LIN {X 0,Y 323.543,Z 923.96,A -85,B 0,C 180,E1 -15317.195,E2 -15317.195} C_VEL
LIN {X 0,Y 320.195,Z 901.46,A -85,B 0,C 180,E1 -15318.02,E2 -15318.02} C_VEL
LIN {X 0,Y 319.838,Z 896.268,A -85,B 0,C 180,E1 -15319.913,E2 -15319.913} C_VEL
LIN {X 0,Y 319.734,Z 895.469,A -85,B 0,C 180,E1 -15320.255,E2 -15320.255} C_VEL
LIN {X 0,Y 319.527,Z 895.494,A -85,B 0,C 180,E1 -15324.703,E2 -15324.703} C_VEL
LIN {X 0,Y 319.569,Z 895.487,A -85,B 0,C 180,E1 -15328.396,E2 -15328.396} C_VEL
LIN {X 0,Y 319.525,Z 895.494,A -85,B 0,C 180,E1 -15331.863,E2 -15331.863} C_VEL
LIN {X 0,Y 319.58,Z 895.491,A -85,B 0,C 180,E1 -15335.543,E2 -15335.543} C_VEL
LIN {X 0,Y 319.53,Z 895.497,A -85,B 0,C 180,E1 -15339.663,E2 -15339.663} C_VEL
LIN {X 0,Y 319.52,Z 895.495,A -85,B 0,C 180,E1 -15343.46,E2 -15343.46} C_VEL
LIN {X 0,Y 319.552,Z 895.489,A -85,B 0,C 180,E1 -15347.016,E2 -15347.016} C_VEL
LIN {X 0,Y 319.517,Z 895.498,A -85,B 0,C 180,E1 -15350.367,E2 -15350.367} C_VEL
LIN {X 0,Y 319.581,Z 895.491,A -85,B 0,C 180,E1 -15354.458,E2 -15354.458} C_VEL
LIN {X 0,Y 319.527,Z 895.494,A -85,B 0,C 180,E1 -15358.138,E2 -15358.138} C_VEL
LIN {X 0,Y 319.572,Z 895.486,A -85,B 0,C 180,E1 -15361.605,E2 -15361.605} C_VEL
LIN {X 0,Y 319.574,Z 895.488,A -85,B 0,C 180,E1 -15365.302,E2 -15365.302} C_VEL
LIN {X 0,Y 319.566,Z 895.487,A -85,B 0,C 180,E1 -15368.046,E2 -15368.046} C_VEL
LIN {X 0,Y 319.596,Z 895.483,A -85,B 0,C 180,E1 -15372.07,E2 -15372.07} C_VEL
LIN {X 0,Y 319.734,Z 895.467,A -85,B 0,C 180,E1 -15376.008,E2 -15376.008} C_VEL
LIN {X 0,Y 319.737,Z 895.469,A -85,B 0,C 180,E1 -15379.872,E2 -15379.872} C_VEL
LIN {X 0,Y 319.901,Z 895.452,A -85,B 0,C 180,E1 -15383.694,E2 -15383.694} C_VEL
LIN {X 0,Y 319.999,Z 895.433,A -85,B 0,C 180,E1 -15388.742,E2 -15388.742} C_VEL
LIN {X 0,Y 319.934,Z 895.444,A -85,B 0,C 180,E1 -15392.518,E2 -15392.518} C_VEL
LIN {X 0,Y 319.901,Z 895.452,A -85,B 0,C 180,E1 -15396.307,E2 -15396.307} C_VEL
LIN {X 0,Y 319.738,Z 895.469,A -85,B 0,C 180,E1 -15400.128,E2 -15400.128} C_VEL
LIN {X 0,Y 319.705,Z 895.471,A -85,B 0,C 180,E1 -15403.994,E2 -15403.994} C_VEL
LIN {X 0,Y 319.589,Z 895.484,A -85,B 0,C 180,E1 -15407.931,E2 -15407.931} C_VEL
LIN {X 0,Y 319.567,Z 895.487,A -85,B 0,C 180,E1 -15411.955,E2 -15411.955} C_VEL
LIN {X 0,Y 319.553,Z 895.489,A -85,B 0,C 180,E1 -15416.096,E2 -15416.096} C_VEL
LIN {X 0,Y 319.544,Z 895.493,A -85,B 0,C 180,E1 -15418.938,E2 -15418.938} C_VEL
LIN {X 0,Y 319.528,Z 895.494,A -85,B 0,C 180,E1 -15421.863,E2 -15421.863} C_VEL
LIN {X 0,Y 319.583,Z 895.491,A -85,B 0,C 180,E1 -15425.542,E2 -15425.542} C_VEL
LIN {X 0,Y 319.532,Z 895.497,A -85,B 0,C 180,E1 -15429.662,E2 -15429.662} C_VEL
LIN {X 0,Y 319.522,Z 895.494,A -85,B 0,C 180,E1 -15433.46,E2 -15433.46} C_VEL
LIN {X 0,Y 319.554,Z 895.489,A -85,B 0,C 180,E1 -15437.015,E2 -15437.015} C_VEL
LIN {X 0,Y 319.518,Z 895.498,A -85,B 0,C 180,E1 -15440.366,E2 -15440.366} C_VEL
LIN {X 0,Y 319.582,Z 895.491,A -85,B 0,C 180,E1 -15444.457,E2 -15444.457} C_VEL
LIN {X 0,Y 319.528,Z 895.494,A -85,B 0,C 180,E1 -15448.137,E2 -15448.137} C_VEL
LIN {X 0,Y 319.572,Z 895.486,A -85,B 0,C 180,E1 -15451.604,E2 -15451.604} C_VEL
LIN {X 0,Y 319.529,Z 895.494,A -85,B 0,C 180,E1 -15455.297,E2 -15455.297} C_VEL
LIN {X 0,Y 319.565,Z 895.487,A -85,B 0,C 180,E1 -15458.045,E2 -15458.045} C_VEL
LIN {X 0,Y 319.552,Z 895.489,A -85,B 0,C 180,E1 -15460.098,E2 -15460.098} C_VEL
LIN {X 0,Y 318.924,Z 895.573,A -85,B 0,C 180,E1 -15461.149,E2 -15461.149} C_VEL
LIN {X 0,Y 316.172,Z 895.918,A -85,B 0,C 180,E1 -15462.862,E2 -15462.862} C_VEL
LIN {X 0,Y 313.804,Z 896.215,A -85,B 0,C 180,E1 -15464.25,E2 -15464.25} C_VEL
LIN {X 0,Y 312.75,Z 896.342,A -85,B 0,C 180,E1 -15465.323,E2 -15465.323} C_VEL
LIN {X 0,Y 312.644,Z 896.352,A -85,B 0,C 180,E1 -15465.686,E2 -15465.686} C_VEL
LIN {X 0,Y 312.686,Z 896.349,A -85,B 0,C 180,E1 -15469.641,E2 -15469.641} C_VEL
LIN {X 0,Y 312.798,Z 896.331,A -85,B 0,C 180,E1 -15472.252,E2 -15472.252} C_VEL
LIN {X 0,Y 312.682,Z 896.345,A -85,B 0,C 180,E1 -15474.841,E2 -15474.841} C_VEL
LIN {X 0,Y 312.965,Z 896.31,A -85,B 0,C 180,E1 -15478.713,E2 -15478.713} C_VEL
LIN {X 0,Y 312.965,Z 896.31,A -85,B 0,C 180,E1 -15481.286,E2 -15481.286} C_VEL
LIN {X 0,Y 312.841,Z 896.329,A -85,B 0,C 180,E1 -15486.449,E2 -15486.449} C_VEL
LIN {X 0,Y 312.752,Z 896.337,A -85,B 0,C 180,E1 -15489.05,E2 -15489.05} C_VEL
LIN {X 0,Y 312.618,Z 896.355,A -85,B 0,C 180,E1 -15492.991,E2 -15492.991} C_VEL
LIN {X 0,Y 312.551,Z 896.361,A -85,B 0,C 180,E1 -15495.654,E2 -15495.654} C_VEL
LIN {X 0,Y 312.529,Z 896.364,A -85,B 0,C 180,E1 -15499.713,E2 -15499.713} C_VEL
LIN {X 0,Y 312.515,Z 896.369,A -85,B 0,C 180,E1 -15502.774,E2 -15502.774} C_VEL
LIN {X 0,Y 312.483,Z 896.371,A -85,B 0,C 180,E1 -15506.731,E2 -15506.731} C_VEL
LIN {X 0,Y 312.494,Z 896.371,A -85,B 0,C 180,E1 -15509.655,E2 -15509.655} C_VEL
LIN {X 0,Y 312.52,Z 896.369,A -85,B 0,C 180,E1 -15513.688,E2 -15513.688} C_VEL
LIN {X 0,Y 312.51,Z 896.369,A -85,B 0,C 180,E1 -15517.387,E2 -15517.387} C_VEL
LIN {X 0,Y 312.44,Z 896.375,A -85,B 0,C 180,E1 -15520.717,E2 -15520.717} C_VEL
LIN {X 0,Y 312.449,Z 896.377,A -85,B 0,C 180,E1 -15524.209,E2 -15524.209} C_VEL
LIN {X 0,Y 312.453,Z 896.377,A -85,B 0,C 180,E1 -15527.924,E2 -15527.924} C_VEL
LIN {X 0,Y 312.475,Z 896.373,A -85,B 0,C 180,E1 -15531.924,E2 -15531.924} C_VEL
LIN {X 0,Y 312.529,Z 896.368,A -85,B 0,C 180,E1 -15534.22,E2 -15534.22} C_VEL
LIN {X 0,Y 312.5,Z 896.368,A -85,B 0,C 180,E1 -15537.333,E2 -15537.333} C_VEL
LIN {X 0,Y 312.518,Z 896.366,A -85,B 0,C 180,E1 -15541.287,E2 -15541.287} C_VEL
LIN {X 0,Y 312.548,Z 896.435,A -85,B 0,C 180,E1 -15542.232,E2 -15542.232} C_VEL
LIN {X 0,Y 314.68,Z 907.796,A -85,B 0,C 180,E1 -15545.947,E2 -15545.947} C_VEL
LIN {X 0,Y 314.406,Z 913.332,A -85,B 0,C 180,E1 -15547.666,E2 -15547.666} C_VEL
LIN {X 0,Y 313.042,Z 926.484,A -85,B 0,C 180,E1 -15551.681,E2 -15551.681} C_VEL
LIN {X 0,Y 315.565,Z 953.099,A -85,B 0,C 180,E1 -15552.654,E2 -15552.654} C_VEL
LIN {X 0,Y 316.221,Z 960.83,A -85,B 0,C 180,E1 -15552.922,E2 -15552.922} C_VEL
LIN {X 0,Y 315.156,Z 1005.028,A -85,B 0,C 180,E1 -15554.354,E2 -15554.354} C_VEL
LIN {X 0,Y 314.521,Z 1016.656,A -85,B 0,C 180,E1 -15554.944,E2 -15554.944} C_VEL
LIN {X 0,Y 314.055,Z 1027.357,A -85,B 0,C 180,E1 -15555.749,E2 -15555.749} C_VEL
LIN {X 0,Y 313.504,Z 1035.704,A -85,B 0,C 180,E1 -15556.551,E2 -15556.551} C_VEL
LIN {X 0,Y 312.921,Z 1043.861,A -85,B 0,C 180,E1 -15557.515,E2 -15557.515} C_VEL
LIN {X 0,Y 312.416,Z 1051.709,A -85,B 0,C 180,E1 -15558.648,E2 -15558.648} C_VEL
LIN {X 0,Y 311.755,Z 1060.752,A -85,B 0,C 180,E1 -15560.266,E2 -15560.266} C_VEL
LIN {X 0,Y 311.364,Z 1067.748,A -85,B 0,C 180,E1 -15561.89,E2 -15561.89} C_VEL
LIN {X 0,Y 311.213,Z 1071.329,A -85,B 0,C 180,E1 -15562.865,E2 -15562.865} C_VEL
LIN {X 0,Y 310.95,Z 1076.877,A -85,B 0,C 180,E1 -15564.813,E2 -15564.813} C_VEL
LIN {X 0,Y 310.886,Z 1079.747,A -85,B 0,C 180,E1 -15566.111,E2 -15566.111} C_VEL
LIN {X 0,Y 310.76,Z 1081.981,A -85,B 0,C 180,E1 -15567.407,E2 -15567.407} C_VEL
LIN {X 0,Y 310.81,Z 1083.616,A -85,B 0,C 180,E1 -15568.704,E2 -15568.704} C_VEL
LIN {X 0,Y 310.844,Z 1084.603,A -85,B 0,C 180,E1 -15570,E2 -15570} C_VEL
LIN {X 0,Y 310.716,Z 1085.026,A -85,B 0,C 180,E1 -15571.296,E2 -15571.296} C_VEL
LIN {X 0,Y 310.723,Z 1084.938,A -85,B 0,C 180,E1 -15572.593,E2 -15572.593} C_VEL
LIN {X 0,Y 310.798,Z 1084.329,A -85,B 0,C 180,E1 -15573.89,E2 -15573.89} C_VEL
LIN {X 0,Y 310.844,Z 1083.162,A -85,B 0,C 180,E1 -15575.189,E2 -15575.189} C_VEL
LIN {X 0,Y 311.156,Z 1080.283,A -85,B 0,C 180,E1 -15577.136,E2 -15577.136} C_VEL
LIN {X 0,Y 311.503,Z 1077.699,A -85,B 0,C 180,E1 -15578.433,E2 -15578.433} C_VEL
LIN {X 0,Y 312.27,Z 1072.48,A -85,B 0,C 180,E1 -15580.372,E2 -15580.372} C_VEL
LIN {X 0,Y 313.209,Z 1066.895,A -85,B 0,C 180,E1 -15581.979,E2 -15581.979} C_VEL
LIN {X 0,Y 314.1,Z 1061.453,A -85,B 0,C 180,E1 -15583.258,E2 -15583.258} C_VEL
LIN {X 0,Y 315.153,Z 1055.012,A -85,B 0,C 180,E1 -15584.529,E2 -15584.529} C_VEL
LIN {X 0,Y 316.58,Z 1046.25,A -85,B 0,C 180,E1 -15585.945,E2 -15585.945} C_VEL
LIN {X 0,Y 318.051,Z 1036.406,A -85,B 0,C 180,E1 -15587.19,E2 -15587.19} C_VEL
LIN {X 0,Y 319.351,Z 1027.107,A -85,B 0,C 180,E1 -15588.11,E2 -15588.11} C_VEL
LIN {X 0,Y 320.71,Z 1016.257,A -85,B 0,C 180,E1 -15588.941,E2 -15588.941} C_VEL
LIN {X 0,Y 321.949,Z 1003.482,A -85,B 0,C 180,E1 -15589.641,E2 -15589.641} C_VEL
LIN {X 0,Y 324.342,Z 961.027,A -85,B 0,C 180,E1 -15591.196,E2 -15591.196} C_VEL
LIN {X 0,Y 323.395,Z 950.536,A -85,B 0,C 180,E1 -15591.773,E2 -15591.773} C_VEL
LIN {X 0,Y 321.025,Z 937.698,A -85,B 0,C 180,E1 -15592.691,E2 -15592.691} C_VEL
LIN {X 0,Y 317.749,Z 924.997,A -85,B 0,C 180,E1 -15593.785,E2 -15593.785} C_VEL
LIN {X 0,Y 317.23,Z 922.474,A -85,B 0,C 180,E1 -15594.046,E2 -15594.046} C_VEL
LIN {X 0,Y 317.491,Z 920.258,A -85,B 0,C 180,E1 -15594.871,E2 -15594.871} C_VEL
LIN {X 0,Y 316.998,Z 915.521,A -85,B 0,C 180,E1 -15596.87,E2 -15596.87} C_VEL
LIN {X 0,Y 315.807,Z 909.438,A -85,B 0,C 180,E1 -15599.784,E2 -15599.784} C_VEL
LIN {X 0,Y 314.73,Z 904.715,A -85,B 0,C 180,E1 -15602.407,E2 -15602.407} C_VEL
LIN {X 0,Y 313.458,Z 899.875,A -85,B 0,C 180,E1 -15605.658,E2 -15605.658} C_VEL
LIN {X 0,Y 312.455,Z 896.377,A -85,B 0,C 180,E1 -15608.768,E2 -15608.768} C_VEL
LIN {X 0,Y 312.462,Z 896.375,A -85,B 0,C 180,E1 -15612.436,E2 -15612.436} C_VEL
LIN {X 0,Y 312.454,Z 896.378,A -85,B 0,C 180,E1 -15616.036,E2 -15616.036} C_VEL
LIN {X 0,Y 312.452,Z 896.377,A -85,B 0,C 180,E1 -15619.886,E2 -15619.886} C_VEL
LIN {X 0,Y 312.531,Z 896.367,A -85,B 0,C 180,E1 -15624.051,E2 -15624.051} C_VEL
LIN {X 0,Y 312.513,Z 896.575,A -85,B 0,C 180,E1 -15627.714,E2 -15627.714} C_VEL
LIN {X 0,Y 313.46,Z 900.147,A -85,B 0,C 180,E1 -15630.975,E2 -15630.975} C_VEL
LIN {X 0,Y 314.53,Z 904.49,A -85,B 0,C 180,E1 -15634.179,E2 -15634.179} C_VEL
LIN {X 0,Y 315.057,Z 906.913,A -85,B 0,C 180,E1 -15635.727,E2 -15635.727} C_VEL
LIN {X 0,Y 317.021,Z 910.62,A -85,B 0,C 180,E1 -15636.252,E2 -15636.252} C_VEL
LIN {X 0,Y 321.671,Z 919.244,A -85,B 0,C 180,E1 -15637.405,E2 -15637.405} C_VEL
LIN {X 0,Y 324.864,Z 926.657,A -85,B 0,C 180,E1 -15638.204,E2 -15638.204} C_VEL
LIN {X 0,Y 325.806,Z 931.165,A -85,B 0,C 180,E1 -15638.542,E2 -15638.542} C_VEL
LIN {X 0,Y 322.501,Z 983.778,A -85,B 0,C 180,E1 -15640.466,E2 -15640.466} C_VEL
LIN {X 0,Y 321.5,Z 996.066,A -85,B 0,C 180,E1 -15641.19,E2 -15641.19} C_VEL
LIN {X 0,Y 320.42,Z 1005.58,A -85,B 0,C 180,E1 -15641.953,E2 -15641.953} C_VEL
LIN {X 0,Y 319.357,Z 1014.7,A -85,B 0,C 180,E1 -15642.883,E2 -15642.883} C_VEL
LIN {X 0,Y 318.001,Z 1024.422,A -85,B 0,C 180,E1 -15644.128,E2 -15644.128} C_VEL
LIN {X 0,Y 316.598,Z 1032.945,A -85,B 0,C 180,E1 -15645.539,E2 -15645.539} C_VEL
LIN {X 0,Y 315.527,Z 1039.167,A -85,B 0,C 180,E1 -15646.803,E2 -15646.803} C_VEL
LIN {X 0,Y 314.468,Z 1044.376,A -85,B 0,C 180,E1 -15648.07,E2 -15648.07} C_VEL
LIN {X 0,Y 313.505,Z 1049.692,A -85,B 0,C 180,E1 -15649.669,E2 -15649.669} C_VEL
LIN {X 0,Y 312.868,Z 1053.097,A -85,B 0,C 180,E1 -15650.954,E2 -15650.954} C_VEL
LIN {X 0,Y 312.03,Z 1057.011,A -85,B 0,C 180,E1 -15652.885,E2 -15652.885} C_VEL
LIN {X 0,Y 311.347,Z 1059.611,A -85,B 0,C 180,E1 -15654.82,E2 -15654.82} C_VEL
LIN {X 0,Y 311.155,Z 1060.559,A -85,B 0,C 180,E1 -15656.115,E2 -15656.115} C_VEL
LIN {X 0,Y 311.003,Z 1060.985,A -85,B 0,C 180,E1 -15657.41,E2 -15657.41} C_VEL
LIN {X 0,Y 310.85,Z 1060.908,A -85,B 0,C 180,E1 -15658.705,E2 -15658.705} C_VEL
LIN {X 0,Y 310.762,Z 1060.312,A -85,B 0,C 180,E1 -15660.001,E2 -15660.001} C_VEL
LIN {X 0,Y 310.739,Z 1059.161,A -85,B 0,C 180,E1 -15661.297,E2 -15661.297} C_VEL
LIN {X 0,Y 310.865,Z 1056.274,A -85,B 0,C 180,E1 -15663.241,E2 -15663.241} C_VEL
LIN {X 0,Y 311,Z 1053.661,A -85,B 0,C 180,E1 -15664.537,E2 -15664.537} C_VEL
LIN {X 0,Y 311.199,Z 1048.47,A -85,B 0,C 180,E1 -15666.446,E2 -15666.446} C_VEL
LIN {X 0,Y 311.597,Z 1042.662,A -85,B 0,C 180,E1 -15668.104,E2 -15668.104} C_VEL
LIN {X 0,Y 312.026,Z 1035.561,A -85,B 0,C 180,E1 -15669.726,E2 -15669.726} C_VEL
LIN {X 0,Y 312.752,Z 1026.431,A -85,B 0,C 180,E1 -15671.34,E2 -15671.34} C_VEL
LIN {X 0,Y 313.268,Z 1018.512,A -85,B 0,C 180,E1 -15672.471,E2 -15672.471} C_VEL
LIN {X 0,Y 313.806,Z 1010.249,A -85,B 0,C 180,E1 -15673.437,E2 -15673.437} C_VEL
LIN {X 0,Y 314.406,Z 998.961,A -85,B 0,C 180,E1 -15674.483,E2 -15674.483} C_VEL
LIN {X 0,Y 314.805,Z 988.035,A -85,B 0,C 180,E1 -15675.208,E2 -15675.208} C_VEL
LIN {X 0,Y 315.175,Z 977.843,A -85,B 0,C 180,E1 -15675.687,E2 -15675.687} C_VEL
LIN {X 0,Y 316.465,Z 924.322,A -85,B 0,C 180,E1 -15677.39,E2 -15677.39} C_VEL
LIN {X 0,Y 313.156,Z 901.751,A -85,B 0,C 180,E1 -15678.234,E2 -15678.234} C_VEL
LIN {X 0,Y 312.683,Z 896.348,A -85,B 0,C 180,E1 -15680.303,E2 -15680.303} C_VEL
LIN {X 0,Y 312.463,Z 896.372,A -85,B 0,C 180,E1 -15683.883,E2 -15683.883} C_VEL
LIN {X 0,Y 312.483,Z 896.371,A -85,B 0,C 180,E1 -15686.733,E2 -15686.733} C_VEL
LIN {X 0,Y 312.495,Z 896.37,A -85,B 0,C 180,E1 -15689.656,E2 -15689.656} C_VEL
LIN {X 0,Y 312.521,Z 896.369,A -85,B 0,C 180,E1 -15693.689,E2 -15693.689} C_VEL
LIN {X 0,Y 312.512,Z 896.369,A -85,B 0,C 180,E1 -15697.388,E2 -15697.388} C_VEL
LIN {X 0,Y 312.442,Z 896.374,A -85,B 0,C 180,E1 -15700.718,E2 -15700.718} C_VEL
LIN {X 0,Y 312.452,Z 896.377,A -85,B 0,C 180,E1 -15704.211,E2 -15704.211} C_VEL
LIN {X 0,Y 312.456,Z 896.377,A -85,B 0,C 180,E1 -15707.926,E2 -15707.926} C_VEL
LIN {X 0,Y 312.478,Z 896.372,A -85,B 0,C 180,E1 -15711.925,E2 -15711.925} C_VEL
LIN {X 0,Y 312.533,Z 896.367,A -85,B 0,C 180,E1 -15714.221,E2 -15714.221} C_VEL
LIN {X 0,Y 312.504,Z 896.367,A -85,B 0,C 180,E1 -15717.334,E2 -15717.334} C_VEL
LIN {X 0,Y 312.507,Z 896.368,A -85,B 0,C 180,E1 -15721.293,E2 -15721.293} C_VEL
LIN {X 0,Y 312.549,Z 896.366,A -85,B 0,C 180,E1 -15724.708,E2 -15724.708} C_VEL
LIN {X 0,Y 312.544,Z 896.363,A -85,B 0,C 180,E1 -15727.526,E2 -15727.526} C_VEL
LIN {X 0,Y 312.557,Z 896.362,A -85,B 0,C 180,E1 -15731.652,E2 -15731.652} C_VEL
LIN {X 0,Y 312.688,Z 896.346,A -85,B 0,C 180,E1 -15735.686,E2 -15735.686} C_VEL
LIN {X 0,Y 312.688,Z 896.349,A -85,B 0,C 180,E1 -15739.642,E2 -15739.642} C_VEL
LIN {X 0,Y 312.8,Z 896.331,A -85,B 0,C 180,E1 -15742.253,E2 -15742.253} C_VEL
LIN {X 0,Y 312.685,Z 896.344,A -85,B 0,C 180,E1 -15744.842,E2 -15744.842} C_VEL
LIN {X 0,Y 312.967,Z 896.31,A -85,B 0,C 180,E1 -15748.713,E2 -15748.713} C_VEL
LIN {X 0,Y 312.967,Z 896.31,A -85,B 0,C 180,E1 -15751.287,E2 -15751.287} C_VEL
LIN {X 0,Y 312.843,Z 896.329,A -85,B 0,C 180,E1 -15756.45,E2 -15756.45} C_VEL
LIN {X 0,Y 312.755,Z 896.336,A -85,B 0,C 180,E1 -15759.05,E2 -15759.05} C_VEL
LIN {X 0,Y 312.621,Z 896.354,A -85,B 0,C 180,E1 -15762.992,E2 -15762.992} C_VEL
LIN {X 0,Y 312.554,Z 896.36,A -85,B 0,C 180,E1 -15765.654,E2 -15765.654} C_VEL
LIN {X 0,Y 312.533,Z 896.363,A -85,B 0,C 180,E1 -15769.713,E2 -15769.713} C_VEL
LIN {X 0,Y 312.519,Z 896.369,A -85,B 0,C 180,E1 -15772.775,E2 -15772.775} C_VEL
LIN {X 0,Y 312.487,Z 896.371,A -85,B 0,C 180,E1 -15776.732,E2 -15776.732} C_VEL
LIN {X 0,Y 312.498,Z 896.37,A -85,B 0,C 180,E1 -15779.655,E2 -15779.655} C_VEL
LIN {X 0,Y 312.524,Z 896.368,A -85,B 0,C 180,E1 -15783.689,E2 -15783.689} C_VEL
LIN {X 0,Y 312.514,Z 896.369,A -85,B 0,C 180,E1 -15787.387,E2 -15787.387} C_VEL
LIN {X 0,Y 312.444,Z 896.374,A -85,B 0,C 180,E1 -15790.717,E2 -15790.717} C_VEL
LIN {X 0,Y 312.454,Z 896.377,A -85,B 0,C 180,E1 -15794.21,E2 -15794.21} C_VEL
LIN {X 0,Y 312.458,Z 896.377,A -85,B 0,C 180,E1 -15797.925,E2 -15797.925} C_VEL
LIN {X 0,Y 312.479,Z 896.372,A -85,B 0,C 180,E1 -15801.924,E2 -15801.924} C_VEL
LIN {X 0,Y 312.534,Z 896.367,A -85,B 0,C 180,E1 -15804.22,E2 -15804.22} C_VEL
LIN {X 0,Y 312.505,Z 896.367,A -85,B 0,C 180,E1 -15807.333,E2 -15807.333} C_VEL
LIN {X 0,Y 312.508,Z 896.367,A -85,B 0,C 180,E1 -15811.292,E2 -15811.292} C_VEL
LIN {X 0,Y 312.52,Z 896.369,A -85,B 0,C 180,E1 -15814.704,E2 -15814.704} C_VEL
LIN {X 0,Y 312.542,Z 896.363,A -85,B 0,C 180,E1 -15817.525,E2 -15817.525} C_VEL
LIN {X 0,Y 312.549,Z 896.363,A -85,B 0,C 180,E1 -15821.65,E2 -15821.65} C_VEL
LIN {X 0,Y 312.644,Z 896.352,A -85,B 0,C 180,E1 -15825.686,E2 -15825.686} C_VEL
LIN {X 0,Y 311.946,Z 896.439,A -85,B 0,C 180,E1 -15826.761,E2 -15826.761} C_VEL
LIN {X 0,Y 309.172,Z 896.782,A -85,B 0,C 180,E1 -15828.515,E2 -15828.515} C_VEL
LIN {X 0,Y 306.845,Z 897.075,A -85,B 0,C 180,E1 -15829.937,E2 -15829.937} C_VEL
LIN {X 0,Y 305.839,Z 897.2,A -85,B 0,C 180,E1 -15831.035,E2 -15831.035} C_VEL
LIN {X 0,Y 305.75,Z 897.21,A -85,B 0,C 180,E1 -15831.407,E2 -15831.407} C_VEL
LIN {X 0,Y 305.787,Z 897.207,A -85,B 0,C 180,E1 -15833.401,E2 -15833.401} C_VEL
LIN {X 0,Y 305.933,Z 897.185,A -85,B 0,C 180,E1 -15838.683,E2 -15838.683} C_VEL
LIN {X 0,Y 305.933,Z 897.186,A -85,B 0,C 180,E1 -15841.316,E2 -15841.316} C_VEL
LIN {X 0,Y 305.786,Z 897.206,A -85,B 0,C 180,E1 -15846.598,E2 -15846.598} C_VEL
LIN {X 0,Y 305.696,Z 897.215,A -85,B 0,C 180,E1 -15849.26,E2 -15849.26} C_VEL
LIN {X 0,Y 305.564,Z 897.232,A -85,B 0,C 180,E1 -15853.297,E2 -15853.297} C_VEL
LIN {X 0,Y 305.498,Z 897.24,A -85,B 0,C 180,E1 -15856.025,E2 -15856.025} C_VEL
LIN {X 0,Y 305.477,Z 897.243,A -85,B 0,C 180,E1 -15860.187,E2 -15860.187} C_VEL
LIN {X 0,Y 305.44,Z 897.247,A -85,B 0,C 180,E1 -15864.466,E2 -15864.466} C_VEL
LIN {X 0,Y 305.449,Z 897.25,A -85,B 0,C 180,E1 -15867.398,E2 -15867.398} C_VEL
LIN {X 0,Y 305.429,Z 897.248,A -85,B 0,C 180,E1 -15870.412,E2 -15870.412} C_VEL
LIN {X 0,Y 305.464,Z 897.244,A -85,B 0,C 180,E1 -15874.078,E2 -15874.078} C_VEL
LIN {X 0,Y 305.451,Z 897.245,A -85,B 0,C 180,E1 -15876.742,E2 -15876.742} C_VEL
LIN {X 0,Y 305.408,Z 897.251,A -85,B 0,C 180,E1 -15880.589,E2 -15880.589} C_VEL
LIN {X 0,Y 305.42,Z 897.252,A -85,B 0,C 180,E1 -15883.656,E2 -15883.656} C_VEL
LIN {X 0,Y 305.433,Z 897.248,A -85,B 0,C 180,E1 -15887.418,E2 -15887.418} C_VEL
LIN {X 0,Y 305.44,Z 897.247,A -85,B 0,C 180,E1 -15891.592,E2 -15891.592} C_VEL
LIN {X 0,Y 305.46,Z 897.246,A -85,B 0,C 180,E1 -15894.886,E2 -15894.886} C_VEL
LIN {X 0,Y 305.44,Z 897.251,A -85,B 0,C 180,E1 -15898.358,E2 -15898.358} C_VEL
LIN {X 0,Y 305.526,Z 897.348,A -85,B 0,C 180,E1 -15902.144,E2 -15902.144} C_VEL
LIN {X 0,Y 307.537,Z 908,A -85,B 0,C 180,E1 -15905.71,E2 -15905.71} C_VEL
LIN {X 0,Y 307.534,Z 912.451,A -85,B 0,C 180,E1 -15907.139,E2 -15907.139} C_VEL
LIN {X 0,Y 305.994,Z 926.268,A -85,B 0,C 180,E1 -15911.46,E2 -15911.46} C_VEL
LIN {X 0,Y 308.607,Z 954.219,A -85,B 0,C 180,E1 -15912.501,E2 -15912.501} C_VEL
LIN {X 0,Y 309.215,Z 960.585,A -85,B 0,C 180,E1 -15912.729,E2 -15912.729} C_VEL
LIN {X 0,Y 308.087,Z 1005.55,A -85,B 0,C 180,E1 -15914.24,E2 -15914.24} C_VEL
LIN {X 0,Y 307.341,Z 1017.878,A -85,B 0,C 180,E1 -15914.923,E2 -15914.923} C_VEL
LIN {X 0,Y 307.028,Z 1026.42,A -85,B 0,C 180,E1 -15915.585,E2 -15915.585} C_VEL
LIN {X 0,Y 306.359,Z 1036.318,A -85,B 0,C 180,E1 -15916.569,E2 -15916.569} C_VEL
LIN {X 0,Y 305.686,Z 1045.522,A -85,B 0,C 180,E1 -15917.721,E2 -15917.721} C_VEL
LIN {X 0,Y 305.121,Z 1054.02,A -85,B 0,C 180,E1 -15919.045,E2 -15919.045} C_VEL
LIN {X 0,Y 304.569,Z 1062.333,A -85,B 0,C 180,E1 -15920.704,E2 -15920.704} C_VEL
LIN {X 0,Y 304.254,Z 1067.769,A -85,B 0,C 180,E1 -15922.033,E2 -15922.033} C_VEL
LIN {X 0,Y 304.072,Z 1072.282,A -85,B 0,C 180,E1 -15923.364,E2 -15923.364} C_VEL
LIN {X 0,Y 303.884,Z 1075.989,A -85,B 0,C 180,E1 -15924.692,E2 -15924.692} C_VEL
LIN {X 0,Y 303.828,Z 1079.004,A -85,B 0,C 180,E1 -15926.021,E2 -15926.021} C_VEL
LIN {X 0,Y 303.685,Z 1081.344,A -85,B 0,C 180,E1 -15927.347,E2 -15927.347} C_VEL
LIN {X 0,Y 303.725,Z 1083.027,A -85,B 0,C 180,E1 -15928.674,E2 -15928.674} C_VEL
LIN {X 0,Y 303.759,Z 1084.114,A -85,B 0,C 180,E1 -15930,E2 -15930} C_VEL
LIN {X 0,Y 303.63,Z 1084.654,A -85,B 0,C 180,E1 -15931.326,E2 -15931.326} C_VEL
LIN {X 0,Y 303.648,Z 1084.679,A -85,B 0,C 180,E1 -15932.653,E2 -15932.653} C_VEL
LIN {X 0,Y 303.712,Z 1084.174,A -85,B 0,C 180,E1 -15933.981,E2 -15933.981} C_VEL
LIN {X 0,Y 303.83,Z 1082.336,A -85,B 0,C 180,E1 -15935.933,E2 -15935.933} C_VEL
LIN {X 0,Y 304.113,Z 1080.391,A -85,B 0,C 180,E1 -15937.302,E2 -15937.302} C_VEL
LIN {X 0,Y 304.709,Z 1076.321,A -85,B 0,C 180,E1 -15939.291,E2 -15939.291} C_VEL
LIN {X 0,Y 305.717,Z 1070.813,A -85,B 0,C 180,E1 -15941.268,E2 -15941.268} C_VEL
LIN {X 0,Y 306.791,Z 1064.993,A -85,B 0,C 180,E1 -15942.906,E2 -15942.906} C_VEL
LIN {X 0,Y 308.01,Z 1057.77,A -85,B 0,C 180,E1 -15944.536,E2 -15944.536} C_VEL
LIN {X 0,Y 309.475,Z 1049.569,A -85,B 0,C 180,E1 -15945.983,E2 -15945.983} C_VEL
LIN {X 0,Y 310.953,Z 1040.647,A -85,B 0,C 180,E1 -15947.256,E2 -15947.256} C_VEL
LIN {X 0,Y 312.451,Z 1031.151,A -85,B 0,C 180,E1 -15948.355,E2 -15948.355} C_VEL
LIN {X 0,Y 314.173,Z 1019.61,A -85,B 0,C 180,E1 -15949.351,E2 -15949.351} C_VEL
LIN {X 0,Y 315.437,Z 1008.952,A -85,B 0,C 180,E1 -15950.033,E2 -15950.033} C_VEL
LIN {X 0,Y 316.409,Z 997.53,A -85,B 0,C 180,E1 -15950.562,E2 -15950.562} C_VEL
LIN {X 0,Y 318.483,Z 962.211,A -85,B 0,C 180,E1 -15951.883,E2 -15951.883} C_VEL
LIN {X 0,Y 317.757,Z 952.743,A -85,B 0,C 180,E1 -15952.428,E2 -15952.428} C_VEL
LIN {X 0,Y 315.352,Z 939.52,A -85,B 0,C 180,E1 -15953.417,E2 -15953.417} C_VEL
LIN {X 0,Y 312.1,Z 926.285,A -85,B 0,C 180,E1 -15954.625,E2 -15954.625} C_VEL
LIN {X 0,Y 310.748,Z 922.017,A -85,B 0,C 180,E1 -15955.128,E2 -15955.128} C_VEL
LIN {X 0,Y 310.312,Z 917.882,A -85,B 0,C 180,E1 -15956.934,E2 -15956.934} C_VEL
LIN {X 0,Y 309.05,Z 911.344,A -85,B 0,C 180,E1 -15960.216,E2 -15960.216} C_VEL
LIN {X 0,Y 307.902,Z 906.268,A -85,B 0,C 180,E1 -15963.217,E2 -15963.217} C_VEL
LIN {X 0,Y 307.012,Z 902.773,A -85,B 0,C 180,E1 -15965.714,E2 -15965.714} C_VEL
LIN {X 0,Y 306.053,Z 899.487,A -85,B 0,C 180,E1 -15968.671,E2 -15968.671} C_VEL
LIN {X 0,Y 305.402,Z 897.257,A -85,B 0,C 180,E1 -15971.514,E2 -15971.514} C_VEL
LIN {X 0,Y 305.396,Z 897.258,A -85,B 0,C 180,E1 -15974.489,E2 -15974.489} C_VEL
LIN {X 0,Y 305.409,Z 897.255,A -85,B 0,C 180,E1 -15978.138,E2 -15978.138} C_VEL
LIN {X 0,Y 305.439,Z 897.25,A -85,B 0,C 180,E1 -15981.593,E2 -15981.593} C_VEL
LIN {X 0,Y 305.459,Z 897.263,A -85,B 0,C 180,E1 -15984.887,E2 -15984.887} C_VEL
LIN {X 0,Y 306.132,Z 899.903,A -85,B 0,C 180,E1 -15988.149,E2 -15988.149} C_VEL
LIN {X 0,Y 306.992,Z 903.284,A -85,B 0,C 180,E1 -15991.266,E2 -15991.266} C_VEL
LIN {X 0,Y 308.035,Z 907.579,A -85,B 0,C 180,E1 -15994.49,E2 -15994.49} C_VEL
LIN {X 0,Y 310.005,Z 911.14,A -85,B 0,C 180,E1 -15995.07,E2 -15995.07} C_VEL
LIN {X 0,Y 311.316,Z 913.444,A -85,B 0,C 180,E1 -15995.445,E2 -15995.445} C_VEL
LIN {X 0,Y 315.229,Z 920.402,A -85,B 0,C 180,E1 -15996.474,E2 -15996.474} C_VEL
LIN {X 0,Y 319.001,Z 928.553,A -85,B 0,C 180,E1 -15997.473,E2 -15997.473} C_VEL
LIN {X 0,Y 320.061,Z 932.769,A -85,B 0,C 180,E1 -15997.827,E2 -15997.827} C_VEL
LIN {X 0,Y 316.361,Z 985.85,A -85,B 0,C 180,E1 -15999.859,E2 -15999.859} C_VEL
LIN {X 0,Y 315.411,Z 996.926,A -85,B 0,C 180,E1 -16000.559,E2 -16000.559} C_VEL
LIN {X 0,Y 314.167,Z 1007.187,A -85,B 0,C 180,E1 -16001.412,E2 -16001.412} C_VEL
LIN {X 0,Y 312.803,Z 1017.357,A -85,B 0,C 180,E1 -16002.512,E2 -16002.512} C_VEL
LIN {X 0,Y 311.54,Z 1025.38,A -85,B 0,C 180,E1 -16003.622,E2 -16003.622} C_VEL
LIN {X 0,Y 310.207,Z 1032.931,A -85,B 0,C 180,E1 -16004.898,E2 -16004.898} C_VEL
LIN {X 0,Y 309.029,Z 1039.231,A -85,B 0,C 180,E1 -16006.185,E2 -16006.185} C_VEL
LIN {X 0,Y 307.633,Z 1045.676,A -85,B 0,C 180,E1 -16007.801,E2 -16007.801} C_VEL
LIN {X 0,Y 306.614,Z 1050.786,A -85,B 0,C 180,E1 -16009.434,E2 -16009.434} C_VEL
LIN {X 0,Y 305.664,Z 1055.395,A -85,B 0,C 180,E1 -16011.37,E2 -16011.37} C_VEL
LIN {X 0,Y 304.743,Z 1058.672,A -85,B 0,C 180,E1 -16013.379,E2 -16013.379} C_VEL
LIN {X 0,Y 304.308,Z 1060.168,A -85,B 0,C 180,E1 -16014.7,E2 -16014.7} C_VEL
LIN {X 0,Y 304.086,Z 1061.07,A -85,B 0,C 180,E1 -16016.025,E2 -16016.025} C_VEL
LIN {X 0,Y 303.92,Z 1061.371,A -85,B 0,C 180,E1 -16017.35,E2 -16017.35} C_VEL
LIN {X 0,Y 303.762,Z 1061.16,A -85,B 0,C 180,E1 -16018.675,E2 -16018.675} C_VEL
LIN {X 0,Y 303.671,Z 1060.44,A -85,B 0,C 180,E1 -16020.001,E2 -16020.001} C_VEL
LIN {X 0,Y 303.653,Z 1059.201,A -85,B 0,C 180,E1 -16021.327,E2 -16021.327} C_VEL
LIN {X 0,Y 303.796,Z 1056.147,A -85,B 0,C 180,E1 -16023.316,E2 -16023.316} C_VEL
LIN {X 0,Y 303.944,Z 1051.742,A -85,B 0,C 180,E1 -16025.308,E2 -16025.308} C_VEL
LIN {X 0,Y 304.29,Z 1045.784,A -85,B 0,C 180,E1 -16027.299,E2 -16027.299} C_VEL
LIN {X 0,Y 304.669,Z 1039.243,A -85,B 0,C 180,E1 -16028.958,E2 -16028.958} C_VEL
LIN {X 0,Y 305.144,Z 1032.866,A -85,B 0,C 180,E1 -16030.283,E2 -16030.283} C_VEL
LIN {X 0,Y 305.691,Z 1025.144,A -85,B 0,C 180,E1 -16031.606,E2 -16031.606} C_VEL
LIN {X 0,Y 306.249,Z 1016.929,A -85,B 0,C 180,E1 -16032.761,E2 -16032.761} C_VEL
LIN {X 0,Y 306.942,Z 1006.707,A -85,B 0,C 180,E1 -16033.912,E2 -16033.912} C_VEL
LIN {X 0,Y 307.521,Z 996.037,A -85,B 0,C 180,E1 -16034.814,E2 -16034.814} C_VEL
LIN {X 0,Y 307.778,Z 986.372,A -85,B 0,C 180,E1 -16035.437,E2 -16035.437} C_VEL
LIN {X 0,Y 308.266,Z 974.608,A -85,B 0,C 180,E1 -16035.963,E2 -16035.963} C_VEL
LIN {X 0,Y 309.47,Z 925.216,A -85,B 0,C 180,E1 -16037.577,E2 -16037.577} C_VEL
LIN {X 0,Y 306.1,Z 902.011,A -85,B 0,C 180,E1 -16038.47,E2 -16038.47} C_VEL
LIN {X 0,Y 305.632,Z 897.227,A -85,B 0,C 180,E1 -16040.353,E2 -16040.353} C_VEL
LIN {X 0,Y 305.44,Z 897.248,A -85,B 0,C 180,E1 -16044.468,E2 -16044.468} C_VEL
LIN {X 0,Y 305.449,Z 897.25,A -85,B 0,C 180,E1 -16047.399,E2 -16047.399} C_VEL
LIN {X 0,Y 305.43,Z 897.247,A -85,B 0,C 180,E1 -16050.413,E2 -16050.413} C_VEL
LIN {X 0,Y 305.466,Z 897.245,A -85,B 0,C 180,E1 -16054.079,E2 -16054.079} C_VEL
LIN {X 0,Y 305.453,Z 897.245,A -85,B 0,C 180,E1 -16056.743,E2 -16056.743} C_VEL
LIN {X 0,Y 305.411,Z 897.25,A -85,B 0,C 180,E1 -16060.59,E2 -16060.59} C_VEL
LIN {X 0,Y 305.422,Z 897.252,A -85,B 0,C 180,E1 -16063.657,E2 -16063.657} C_VEL
LIN {X 0,Y 305.436,Z 897.248,A -85,B 0,C 180,E1 -16067.419,E2 -16067.419} C_VEL
LIN {X 0,Y 305.443,Z 897.247,A -85,B 0,C 180,E1 -16071.593,E2 -16071.593} C_VEL
LIN {X 0,Y 305.464,Z 897.246,A -85,B 0,C 180,E1 -16074.887,E2 -16074.887} C_VEL
LIN {X 0,Y 305.445,Z 897.249,A -85,B 0,C 180,E1 -16078.359,E2 -16078.359} C_VEL
LIN {X 0,Y 305.477,Z 897.245,A -85,B 0,C 180,E1 -16081.109,E2 -16081.109} C_VEL
LIN {X 0,Y 305.501,Z 897.24,A -85,B 0,C 180,E1 -16084.082,E2 -16084.082} C_VEL
LIN {X 0,Y 305.477,Z 897.248,A -85,B 0,C 180,E1 -16086.976,E2 -16086.976} C_VEL
LIN {X 0,Y 305.513,Z 897.243,A -85,B 0,C 180,E1 -16091.213,E2 -16091.213} C_VEL
LIN {X 0,Y 305.63,Z 897.229,A -85,B 0,C 180,E1 -16095.348,E2 -16095.348} C_VEL
LIN {X 0,Y 305.626,Z 897.228,A -85,B 0,C 180,E1 -16099.4,E2 -16099.4} C_VEL
LIN {X 0,Y 305.75,Z 897.21,A -85,B 0,C 180,E1 -16102.073,E2 -16102.073} C_VEL
LIN {X 0,Y 305.656,Z 897.219,A -85,B 0,C 180,E1 -16104.723,E2 -16104.723} C_VEL
LIN {X 0,Y 305.935,Z 897.186,A -85,B 0,C 180,E1 -16108.684,E2 -16108.684} C_VEL
LIN {X 0,Y 305.935,Z 897.186,A -85,B 0,C 180,E1 -16111.317,E2 -16111.317} C_VEL
LIN {X 0,Y 305.789,Z 897.206,A -85,B 0,C 180,E1 -16116.599,E2 -16116.599} C_VEL
LIN {X 0,Y 305.699,Z 897.215,A -85,B 0,C 180,E1 -16119.261,E2 -16119.261} C_VEL
LIN {X 0,Y 305.567,Z 897.231,A -85,B 0,C 180,E1 -16123.297,E2 -16123.297} C_VEL
LIN {X 0,Y 305.501,Z 897.24,A -85,B 0,C 180,E1 -16126.025,E2 -16126.025} C_VEL
LIN {X 0,Y 305.48,Z 897.242,A -85,B 0,C 180,E1 -16130.188,E2 -16130.188} C_VEL
LIN {X 0,Y 305.444,Z 897.247,A -85,B 0,C 180,E1 -16134.467,E2 -16134.467} C_VEL
LIN {X 0,Y 305.453,Z 897.25,A -85,B 0,C 180,E1 -16137.398,E2 -16137.398} C_VEL
LIN {X 0,Y 305.433,Z 897.247,A -85,B 0,C 180,E1 -16140.413,E2 -16140.413} C_VEL
LIN {X 0,Y 305.469,Z 897.244,A -85,B 0,C 180,E1 -16144.078,E2 -16144.078} C_VEL
LIN {X 0,Y 305.456,Z 897.245,A -85,B 0,C 180,E1 -16146.743,E2 -16146.743} C_VEL
LIN {X 0,Y 305.413,Z 897.25,A -85,B 0,C 180,E1 -16150.589,E2 -16150.589} C_VEL
LIN {X 0,Y 305.424,Z 897.252,A -85,B 0,C 180,E1 -16153.656,E2 -16153.656} C_VEL
LIN {X 0,Y 305.438,Z 897.248,A -85,B 0,C 180,E1 -16157.418,E2 -16157.418} C_VEL
LIN {X 0,Y 305.445,Z 897.246,A -85,B 0,C 180,E1 -16161.592,E2 -16161.592} C_VEL
LIN {X 0,Y 305.465,Z 897.246,A -85,B 0,C 180,E1 -16164.886,E2 -16164.886} C_VEL
LIN {X 0,Y 305.445,Z 897.25,A -85,B 0,C 180,E1 -16168.358,E2 -16168.358} C_VEL
LIN {X 0,Y 305.477,Z 897.244,A -85,B 0,C 180,E1 -16171.109,E2 -16171.109} C_VEL
LIN {X 0,Y 305.482,Z 897.242,A -85,B 0,C 180,E1 -16174.079,E2 -16174.079} C_VEL
LIN {X 0,Y 305.461,Z 897.245,A -85,B 0,C 180,E1 -16178.399,E2 -16178.399} C_VEL
LIN {X 0,Y 305.505,Z 897.244,A -85,B 0,C 180,E1 -16181.212,E2 -16181.212} C_VEL
LIN {X 0,Y 305.555,Z 897.235,A -85,B 0,C 180,E1 -16185.677,E2 -16185.677} C_VEL
LIN {X 0,Y 305.624,Z 897.228,A -85,B 0,C 180,E1 -16189.399,E2 -16189.399} C_VEL
LIN {X 0,Y 305.75,Z 897.21,A -85,B 0,C 180,E1 -16191.407,E2 -16191.407} C_VEL
LIN {X 0,Y 305.029,Z 897.299,A -85,B 0,C 180,E1 -16192.505,E2 -16192.505} C_VEL
LIN {X 0,Y 302.067,Z 897.668,A -85,B 0,C 180,E1 -16194.291,E2 -16194.291} C_VEL
LIN {X 0,Y 299.668,Z 897.971,A -85,B 0,C 180,E1 -16195.74,E2 -16195.74} C_VEL
LIN {X 0,Y 298.775,Z 898.077,A -85,B 0,C 180,E1 -16196.864,E2 -16196.864} C_VEL
LIN {X 0,Y 298.775,Z 898.077,A -85,B 0,C 180,E1 -16197.244,E2 -16197.244} C_VEL
LIN {X 0,Y 298.886,Z 898.069,A -85,B 0,C 180,E1 -16199.999,E2 -16199.999} C_VEL
LIN {X 0,Y 298.788,Z 898.077,A -85,B 0,C 180,E1 -16202.696,E2 -16202.696} C_VEL
LIN {X 0,Y 298.735,Z 898.083,A -85,B 0,C 180,E1 -16206.755,E2 -16206.755} C_VEL
LIN {X 0,Y 298.626,Z 898.096,A -85,B 0,C 180,E1 -16209.482,E2 -16209.482} C_VEL
LIN {X 0,Y 298.517,Z 898.109,A -85,B 0,C 180,E1 -16213.616,E2 -16213.616} C_VEL
LIN {X 0,Y 298.441,Z 898.121,A -85,B 0,C 180,E1 -16216.414,E2 -16216.414} C_VEL
LIN {X 0,Y 298.433,Z 898.12,A -85,B 0,C 180,E1 -16219.611,E2 -16219.611} C_VEL
LIN {X 0,Y 298.382,Z 898.127,A -85,B 0,C 180,E1 -16223.603,E2 -16223.603} C_VEL
LIN {X 0,Y 298.402,Z 898.124,A -85,B 0,C 180,E1 -16226.582,E2 -16226.582} C_VEL
LIN {X 0,Y 298.393,Z 898.128,A -85,B 0,C 180,E1 -16229.643,E2 -16229.643} C_VEL
LIN {X 0,Y 298.393,Z 898.125,A -85,B 0,C 180,E1 -16232.8,E2 -16232.8} C_VEL
LIN {X 0,Y 298.426,Z 898.121,A -85,B 0,C 180,E1 -16236.801,E2 -16236.801} C_VEL
LIN {X 0,Y 298.373,Z 898.131,A -85,B 0,C 180,E1 -16239.491,E2 -16239.491} C_VEL
LIN {X 0,Y 298.369,Z 898.127,A -85,B 0,C 180,E1 -16243.096,E2 -16243.096} C_VEL
LIN {X 0,Y 298.369,Z 898.128,A -85,B 0,C 180,E1 -16246.914,E2 -16246.914} C_VEL
LIN {X 0,Y 298.384,Z 898.126,A -85,B 0,C 180,E1 -16251.01,E2 -16251.01} C_VEL
LIN {X 0,Y 298.403,Z 898.124,A -85,B 0,C 180,E1 -16253.928,E2 -16253.928} C_VEL
LIN {X 0,Y 298.392,Z 898.126,A -85,B 0,C 180,E1 -16257.199,E2 -16257.199} C_VEL
LIN {X 0,Y 298.507,Z 898.242,A -85,B 0,C 180,E1 -16262.055,E2 -16262.055} C_VEL
LIN {X 0,Y 300.527,Z 909.147,A -85,B 0,C 180,E1 -16265.788,E2 -16265.788} C_VEL
LIN {X 0,Y 300.383,Z 913.75,A -85,B 0,C 180,E1 -16267.291,E2 -16267.291} C_VEL
LIN {X 0,Y 298.973,Z 926.03,A -85,B 0,C 180,E1 -16271.231,E2 -16271.231} C_VEL
LIN {X 0,Y 301.309,Z 952.578,A -85,B 0,C 180,E1 -16272.25,E2 -16272.25} C_VEL
LIN {X 0,Y 302.149,Z 961.305,A -85,B 0,C 180,E1 -16272.578,E2 -16272.578} C_VEL
LIN {X 0,Y 301.031,Z 1005.271,A -85,B 0,C 180,E1 -16274.122,E2 -16274.122} C_VEL
LIN {X 0,Y 300.284,Z 1017.546,A -85,B 0,C 180,E1 -16274.821,E2 -16274.821} C_VEL
LIN {X 0,Y 299.919,Z 1026.985,A -85,B 0,C 180,E1 -16275.583,E2 -16275.583} C_VEL
LIN {X 0,Y 299.33,Z 1035.244,A -85,B 0,C 180,E1 -16276.42,E2 -16276.42} C_VEL
LIN {X 0,Y 298.767,Z 1043.36,A -85,B 0,C 180,E1 -16277.432,E2 -16277.432} C_VEL
LIN {X 0,Y 298.252,Z 1051.176,A -85,B 0,C 180,E1 -16278.618,E2 -16278.618} C_VEL
LIN {X 0,Y 297.648,Z 1059.397,A -85,B 0,C 180,E1 -16280.143,E2 -16280.143} C_VEL
LIN {X 0,Y 297.225,Z 1066.557,A -85,B 0,C 180,E1 -16281.844,E2 -16281.844} C_VEL
LIN {X 0,Y 297.039,Z 1071.243,A -85,B 0,C 180,E1 -16283.206,E2 -16283.206} C_VEL
LIN {X 0,Y 296.824,Z 1075.102,A -85,B 0,C 180,E1 -16284.565,E2 -16284.565} C_VEL
LIN {X 0,Y 296.771,Z 1078.236,A -85,B 0,C 180,E1 -16285.926,E2 -16285.926} C_VEL
LIN {X 0,Y 296.614,Z 1080.632,A -85,B 0,C 180,E1 -16287.284,E2 -16287.284} C_VEL
LIN {X 0,Y 296.643,Z 1082.399,A -85,B 0,C 180,E1 -16288.642,E2 -16288.642} C_VEL
LIN {X 0,Y 296.676,Z 1083.606,A -85,B 0,C 180,E1 -16290,E2 -16290} C_VEL
LIN {X 0,Y 296.546,Z 1084.271,A -85,B 0,C 180,E1 -16291.358,E2 -16291.358} C_VEL
LIN {X 0,Y 296.574,Z 1084.423,A -85,B 0,C 180,E1 -16292.716,E2 -16292.716} C_VEL
LIN {X 0,Y 296.629,Z 1083.963,A -85,B 0,C 180,E1 -16294.076,E2 -16294.076} C_VEL
LIN {X 0,Y 296.735,Z 1082.534,A -85,B 0,C 180,E1 -16295.88,E2 -16295.88} C_VEL
LIN {X 0,Y 297.256,Z 1079.27,A -85,B 0,C 180,E1 -16298.155,E2 -16298.155} C_VEL
LIN {X 0,Y 297.993,Z 1074.984,A -85,B 0,C 180,E1 -16300.188,E2 -16300.188} C_VEL
LIN {X 0,Y 298.979,Z 1070.273,A -85,B 0,C 180,E1 -16301.869,E2 -16301.869} C_VEL
LIN {X 0,Y 300.131,Z 1064.391,A -85,B 0,C 180,E1 -16303.542,E2 -16303.542} C_VEL
LIN {X 0,Y 301.576,Z 1057.095,A -85,B 0,C 180,E1 -16305.199,E2 -16305.199} C_VEL
LIN {X 0,Y 303.148,Z 1048.913,A -85,B 0,C 180,E1 -16306.672,E2 -16306.672} C_VEL
LIN {X 0,Y 304.75,Z 1040.02,A -85,B 0,C 180,E1 -16307.965,E2 -16307.965} C_VEL
LIN {X 0,Y 306.666,Z 1028.866,A -85,B 0,C 180,E1 -16309.234,E2 -16309.234} C_VEL
LIN {X 0,Y 308.309,Z 1017.718,A -85,B 0,C 180,E1 -16310.168,E2 -16310.168} C_VEL
LIN {X 0,Y 309.645,Z 1006.9,A -85,B 0,C 180,E1 -16310.858,E2 -16310.858} C_VEL
LIN {X 0,Y 310.931,Z 991.059,A -85,B 0,C 180,E1 -16311.541,E2 -16311.541} C_VEL
LIN {X 0,Y 312.726,Z 962.922,A -85,B 0,C 180,E1 -16312.635,E2 -16312.635} C_VEL
LIN {X 0,Y 312.042,Z 954.091,A -85,B 0,C 180,E1 -16313.178,E2 -16313.178} C_VEL
LIN {X 0,Y 309.86,Z 941.44,A -85,B 0,C 180,E1 -16314.184,E2 -16314.184} C_VEL
LIN {X 0,Y 307,Z 929.66,A -85,B 0,C 180,E1 -16315.325,E2 -16315.325} C_VEL
LIN {X 0,Y 305.595,Z 925.762,A -85,B 0,C 180,E1 -16315.815,E2 -16315.815} C_VEL
LIN {X 0,Y 303.806,Z 921.574,A -85,B 0,C 180,E1 -16316.406,E2 -16316.406} C_VEL
LIN {X 0,Y 302.876,Z 915.999,A -85,B 0,C 180,E1 -16319.162,E2 -16319.162} C_VEL
LIN {X 0,Y 301.727,Z 910.418,A -85,B 0,C 180,E1 -16322.393,E2 -16322.393} C_VEL
LIN {X 0,Y 300.557,Z 905.693,A -85,B 0,C 180,E1 -16325.773,E2 -16325.773} C_VEL
LIN {X 0,Y 299.453,Z 902.014,A -85,B 0,C 180,E1 -16329.322,E2 -16329.322} C_VEL
LIN {X 0,Y 299.034,Z 900.53,A -85,B 0,C 180,E1 -16331.23,E2 -16331.23} C_VEL
LIN {X 0,Y 298.449,Z 898.667,A -85,B 0,C 180,E1 -16335.054,E2 -16335.054} C_VEL
LIN {X 0,Y 298.401,Z 898.245,A -85,B 0,C 180,E1 -16336.921,E2 -16336.921} C_VEL
LIN {X 0,Y 298.412,Z 898.476,A -85,B 0,C 180,E1 -16340.515,E2 -16340.515} C_VEL
LIN {X 0,Y 298.866,Z 899.794,A -85,B 0,C 180,E1 -16343.993,E2 -16343.993} C_VEL
LIN {X 0,Y 299.541,Z 902.383,A -85,B 0,C 180,E1 -16347.635,E2 -16347.635} C_VEL
LIN {X 0,Y 300.3,Z 905.248,A -85,B 0,C 180,E1 -16350.563,E2 -16350.563} C_VEL
LIN {X 0,Y 301.028,Z 908.427,A -85,B 0,C 180,E1 -16353.088,E2 -16353.088} C_VEL
LIN {X 0,Y 303.101,Z 912.022,A -85,B 0,C 180,E1 -16353.772,E2 -16353.772} C_VEL
LIN {X 0,Y 304.357,Z 913.849,A -85,B 0,C 180,E1 -16354.152,E2 -16354.152} C_VEL
LIN {X 0,Y 308.581,Z 921.068,A -85,B 0,C 180,E1 -16355.38,E2 -16355.38} C_VEL
LIN {X 0,Y 313.269,Z 930.646,A -85,B 0,C 180,E1 -16356.697,E2 -16356.697} C_VEL
LIN {X 0,Y 314.417,Z 934.176,A -85,B 0,C 180,E1 -16357.065,E2 -16357.065} C_VEL
LIN {X 0,Y 310.627,Z 985.174,A -85,B 0,C 180,E1 -16359.081,E2 -16359.081} C_VEL
LIN {X 0,Y 309.457,Z 997.039,A -85,B 0,C 180,E1 -16359.824,E2 -16359.824} C_VEL
LIN {X 0,Y 308.161,Z 1007.186,A -85,B 0,C 180,E1 -16360.69,E2 -16360.69} C_VEL
LIN {X 0,Y 306.717,Z 1017.392,A -85,B 0,C 180,E1 -16361.809,E2 -16361.809} C_VEL
LIN {X 0,Y 305.382,Z 1025.508,A -85,B 0,C 180,E1 -16362.937,E2 -16362.937} C_VEL
LIN {X 0,Y 303.895,Z 1033.097,A -85,B 0,C 180,E1 -16364.233,E2 -16364.233} C_VEL
LIN {X 0,Y 302.587,Z 1039.386,A -85,B 0,C 180,E1 -16365.542,E2 -16365.542} C_VEL
LIN {X 0,Y 301.113,Z 1045.806,A -85,B 0,C 180,E1 -16367.19,E2 -16367.19} C_VEL
LIN {X 0,Y 300.12,Z 1050.025,A -85,B 0,C 180,E1 -16368.519,E2 -16368.519} C_VEL
LIN {X 0,Y 299.32,Z 1053.495,A -85,B 0,C 180,E1 -16369.858,E2 -16369.858} C_VEL
LIN {X 0,Y 298.353,Z 1057.458,A -85,B 0,C 180,E1 -16371.875,E2 -16371.875} C_VEL
LIN {X 0,Y 297.738,Z 1059.345,A -85,B 0,C 180,E1 -16373.223,E2 -16373.223} C_VEL
LIN {X 0,Y 297.273,Z 1060.693,A -85,B 0,C 180,E1 -16374.574,E2 -16374.574} C_VEL
LIN {X 0,Y 297.021,Z 1061.521,A -85,B 0,C 180,E1 -16375.93,E2 -16375.93} C_VEL
LIN {X 0,Y 296.84,Z 1061.755,A -85,B 0,C 180,E1 -16377.287,E2 -16377.287} C_VEL
LIN {X 0,Y 296.676,Z 1061.408,A -85,B 0,C 180,E1 -16378.643,E2 -16378.643} C_VEL
LIN {X 0,Y 296.584,Z 1060.553,A -85,B 0,C 180,E1 -16380.001,E2 -16380.001} C_VEL
LIN {X 0,Y 296.571,Z 1059.169,A -85,B 0,C 180,E1 -16381.359,E2 -16381.359} C_VEL
LIN {X 0,Y 296.728,Z 1055.976,A -85,B 0,C 180,E1 -16383.395,E2 -16383.395} C_VEL
LIN {X 0,Y 296.823,Z 1053.079,A -85,B 0,C 180,E1 -16384.754,E2 -16384.754} C_VEL
LIN {X 0,Y 297.001,Z 1048.781,A -85,B 0,C 180,E1 -16386.355,E2 -16386.355} C_VEL
LIN {X 0,Y 297.335,Z 1043.932,A -85,B 0,C 180,E1 -16387.812,E2 -16387.812} C_VEL
LIN {X 0,Y 297.645,Z 1038.434,A -85,B 0,C 180,E1 -16389.172,E2 -16389.172} C_VEL
LIN {X 0,Y 298.138,Z 1031.834,A -85,B 0,C 180,E1 -16390.527,E2 -16390.527} C_VEL
LIN {X 0,Y 298.805,Z 1022.782,A -85,B 0,C 180,E1 -16392.049,E2 -16392.049} C_VEL
LIN {X 0,Y 299.487,Z 1012.341,A -85,B 0,C 180,E1 -16393.4,E2 -16393.4} C_VEL
LIN {X 0,Y 300.049,Z 1004.267,A -85,B 0,C 180,E1 -16394.238,E2 -16394.238} C_VEL
LIN {X 0,Y 300.506,Z 995.183,A -85,B 0,C 180,E1 -16394.995,E2 -16394.995} C_VEL
LIN {X 0,Y 300.829,Z 983.751,A -85,B 0,C 180,E1 -16395.716,E2 -16395.716} C_VEL
LIN {X 0,Y 301.395,Z 967.863,A -85,B 0,C 180,E1 -16396.325,E2 -16396.325} C_VEL
LIN {X 0,Y 302.407,Z 925.589,A -85,B 0,C 180,E1 -16397.762,E2 -16397.762} C_VEL
LIN {X 0,Y 299.036,Z 902.333,A -85,B 0,C 180,E1 -16398.676,E2 -16398.676} C_VEL
LIN {X 0,Y 298.603,Z 898.099,A -85,B 0,C 180,E1 -16400.356,E2 -16400.356} C_VEL
LIN {X 0,Y 298.414,Z 898.128,A -85,B 0,C 180,E1 -16405.083,E2 -16405.083} C_VEL
LIN {X 0,Y 298.402,Z 898.128,A -85,B 0,C 180,E1 -16409.375,E2 -16409.375} C_VEL
LIN {X 0,Y 298.394,Z 898.125,A -85,B 0,C 180,E1 -16412.801,E2 -16412.801} C_VEL
LIN {X 0,Y 298.428,Z 898.12,A -85,B 0,C 180,E1 -16416.803,E2 -16416.803} C_VEL
LIN {X 0,Y 298.348,Z 898.131,A -85,B 0,C 180,E1 -16421.269,E2 -16421.269} C_VEL
LIN {X 0,Y 298.357,Z 898.129,A -85,B 0,C 180,E1 -16425.035,E2 -16425.035} C_VEL
LIN {X 0,Y 298.349,Z 898.13,A -85,B 0,C 180,E1 -16428.922,E2 -16428.922} C_VEL
LIN {X 0,Y 298.389,Z 898.13,A -85,B 0,C 180,E1 -16432.238,E2 -16432.238} C_VEL
LIN {X 0,Y 298.411,Z 898.122,A -85,B 0,C 180,E1 -16435.582,E2 -16435.582} C_VEL
LIN {X 0,Y 298.38,Z 898.13,A -85,B 0,C 180,E1 -16438.79,E2 -16438.79} C_VEL
LIN {X 0,Y 298.414,Z 898.122,A -85,B 0,C 180,E1 -16441.899,E2 -16441.899} C_VEL
LIN {X 0,Y 298.441,Z 898.124,A -85,B 0,C 180,E1 -16444.92,E2 -16444.92} C_VEL
LIN {X 0,Y 298.401,Z 898.123,A -85,B 0,C 180,E1 -16447.862,E2 -16447.862} C_VEL
LIN {X 0,Y 298.463,Z 898.118,A -85,B 0,C 180,E1 -16450.752,E2 -16450.752} C_VEL
LIN {X 0,Y 298.59,Z 898.103,A -85,B 0,C 180,E1 -16454.995,E2 -16454.995} C_VEL
LIN {X 0,Y 298.585,Z 898.103,A -85,B 0,C 180,E1 -16459.147,E2 -16459.147} C_VEL
LIN {X 0,Y 298.702,Z 898.09,A -85,B 0,C 180,E1 -16461.885,E2 -16461.885} C_VEL
LIN {X 0,Y 298.626,Z 898.095,A -85,B 0,C 180,E1 -16464.599,E2 -16464.599} C_VEL
LIN {X 0,Y 298.902,Z 898.062,A -85,B 0,C 180,E1 -16468.653,E2 -16468.653} C_VEL
LIN {X 0,Y 298.902,Z 898.062,A -85,B 0,C 180,E1 -16471.348,E2 -16471.348} C_VEL
LIN {X 0,Y 298.738,Z 898.083,A -85,B 0,C 180,E1 -16476.756,E2 -16476.756} C_VEL
LIN {X 0,Y 298.629,Z 898.095,A -85,B 0,C 180,E1 -16479.482,E2 -16479.482} C_VEL
LIN {X 0,Y 298.52,Z 898.108,A -85,B 0,C 180,E1 -16483.617,E2 -16483.617} C_VEL
LIN {X 0,Y 298.445,Z 898.121,A -85,B 0,C 180,E1 -16486.415,E2 -16486.415} C_VEL
LIN {X 0,Y 298.436,Z 898.12,A -85,B 0,C 180,E1 -16489.611,E2 -16489.611} C_VEL
LIN {X 0,Y 298.386,Z 898.126,A -85,B 0,C 180,E1 -16493.604,E2 -16493.604} C_VEL
LIN {X 0,Y 298.406,Z 898.124,A -85,B 0,C 180,E1 -16496.583,E2 -16496.583} C_VEL
LIN {X 0,Y 298.397,Z 898.127,A -85,B 0,C 180,E1 -16499.644,E2 -16499.644} C_VEL
LIN {X 0,Y 298.397,Z 898.124,A -85,B 0,C 180,E1 -16502.8,E2 -16502.8} C_VEL
LIN {X 0,Y 298.43,Z 898.12,A -85,B 0,C 180,E1 -16506.802,E2 -16506.802} C_VEL
LIN {X 0,Y 298.378,Z 898.13,A -85,B 0,C 180,E1 -16509.492,E2 -16509.492} C_VEL
LIN {X 0,Y 298.373,Z 898.127,A -85,B 0,C 180,E1 -16513.097,E2 -16513.097} C_VEL
LIN {X 0,Y 298.373,Z 898.127,A -85,B 0,C 180,E1 -16516.914,E2 -16516.914} C_VEL
LIN {X 0,Y 298.388,Z 898.125,A -85,B 0,C 180,E1 -16521.011,E2 -16521.011} C_VEL
LIN {X 0,Y 298.408,Z 898.124,A -85,B 0,C 180,E1 -16523.928,E2 -16523.928} C_VEL
LIN {X 0,Y 298.397,Z 898.125,A -85,B 0,C 180,E1 -16527.199,E2 -16527.199} C_VEL
LIN {X 0,Y 298.405,Z 898.128,A -85,B 0,C 180,E1 -16530.625,E2 -16530.625} C_VEL
LIN {X 0,Y 298.416,Z 898.128,A -85,B 0,C 180,E1 -16534.917,E2 -16534.917} C_VEL
LIN {X 0,Y 298.393,Z 898.124,A -85,B 0,C 180,E1 -16537.861,E2 -16537.861} C_VEL
LIN {X 0,Y 298.456,Z 898.119,A -85,B 0,C 180,E1 -16540.75,E2 -16540.75} C_VEL
LIN {X 0,Y 298.513,Z 898.113,A -85,B 0,C 180,E1 -16544.99,E2 -16544.99} C_VEL
LIN {X 0,Y 298.583,Z 898.103,A -85,B 0,C 180,E1 -16549.146,E2 -16549.146} C_VEL
LIN {X 0,Y 298.701,Z 898.09,A -85,B 0,C 180,E1 -16551.884,E2 -16551.884} C_VEL
LIN {X 0,Y 298.624,Z 898.096,A -85,B 0,C 180,E1 -16554.598,E2 -16554.598} C_VEL
LIN {X 0,Y 298.775,Z 898.077,A -85,B 0,C 180,E1 -16557.244,E2 -16557.244} C_VEL
LIN {X 0,Y 298.315,Z 898.139,A -85,B 0,C 180,E1 -16558.37,E2 -16558.37} C_VEL
LIN {X 0,Y 296.827,Z 898.324,A -85,B 0,C 180,E1 -16559.476,E2 -16559.476} C_VEL
LIN {X 0,Y 293.009,Z 898.798,A -85,B 0,C 180,E1 -16561.691,E2 -16561.691} C_VEL
LIN {X 0,Y 291.796,Z 898.948,A -85,B 0,C 180,E1 -16562.844,E2 -16562.844} C_VEL
LIN {X 0,Y 291.64,Z 898.966,A -85,B 0,C 180,E1 -16563.236,E2 -16563.236} C_VEL
LIN {X 0,Y 291.687,Z 898.96,A -85,B 0,C 180,E1 -16566.919,E2 -16566.919} C_VEL
LIN {X 0,Y 291.569,Z 898.975,A -85,B 0,C 180,E1 -16569.713,E2 -16569.713} C_VEL
LIN {X 0,Y 291.477,Z 898.987,A -85,B 0,C 180,E1 -16573.952,E2 -16573.952} C_VEL
LIN {X 0,Y 291.378,Z 898.999,A -85,B 0,C 180,E1 -16578.273,E2 -16578.273} C_VEL
LIN {X 0,Y 291.342,Z 899.006,A -85,B 0,C 180,E1 -16581.213,E2 -16581.213} C_VEL
LIN {X 0,Y 291.326,Z 899.005,A -85,B 0,C 180,E1 -16584.211,E2 -16584.211} C_VEL
LIN {X 0,Y 291.35,Z 899.007,A -85,B 0,C 180,E1 -16587.278,E2 -16587.278} C_VEL
LIN {X 0,Y 291.318,Z 899.006,A -85,B 0,C 180,E1 -16590.438,E2 -16590.438} C_VEL
LIN {X 0,Y 291.344,Z 899.005,A -85,B 0,C 180,E1 -16593.698,E2 -16593.698} C_VEL
LIN {X 0,Y 291.352,Z 899.004,A -85,B 0,C 180,E1 -16597.247,E2 -16597.247} C_VEL
LIN {X 0,Y 291.299,Z 899.009,A -85,B 0,C 180,E1 -16600.648,E2 -16600.648} C_VEL
LIN {X 0,Y 291.281,Z 899.012,A -85,B 0,C 180,E1 -16604.403,E2 -16604.403} C_VEL
LIN {X 0,Y 291.293,Z 899.013,A -85,B 0,C 180,E1 -16608.411,E2 -16608.411} C_VEL
LIN {X 0,Y 291.332,Z 899.004,A -85,B 0,C 180,E1 -16611.154,E2 -16611.154} C_VEL
LIN {X 0,Y 291.354,Z 899.005,A -85,B 0,C 180,E1 -16614.625,E2 -16614.625} C_VEL
LIN {X 0,Y 291.365,Z 899.001,A -85,B 0,C 180,E1 -16617.949,E2 -16617.949} C_VEL
LIN {X 0,Y 291.472,Z 899.059,A -85,B 0,C 180,E1 -16621.953,E2 -16621.953} C_VEL
LIN {X 0,Y 293.365,Z 909.316,A -85,B 0,C 180,E1 -16625.552,E2 -16625.552} C_VEL
LIN {X 0,Y 293.472,Z 912.78,A -85,B 0,C 180,E1 -16626.725,E2 -16626.725} C_VEL
LIN {X 0,Y 291.95,Z 925.734,A -85,B 0,C 180,E1 -16630.99,E2 -16630.99} C_VEL
LIN {X 0,Y 293.692,Z 947.547,A -85,B 0,C 180,E1 -16631.875,E2 -16631.875} C_VEL
LIN {X 0,Y 295.152,Z 960.582,A -85,B 0,C 180,E1 -16632.387,E2 -16632.387} C_VEL
LIN {X 0,Y 293.976,Z 1004.94,A -85,B 0,C 180,E1 -16633.997,E2 -16633.997} C_VEL
LIN {X 0,Y 293.215,Z 1017.207,A -85,B 0,C 180,E1 -16634.713,E2 -16634.713} C_VEL
LIN {X 0,Y 292.77,Z 1027.529,A -85,B 0,C 180,E1 -16635.578,E2 -16635.578} C_VEL
LIN {X 0,Y 292.083,Z 1037.111,A -85,B 0,C 180,E1 -16636.609,E2 -16636.609} C_VEL
LIN {X 0,Y 291.376,Z 1047.212,A -85,B 0,C 180,E1 -16637.992,E2 -16637.992} C_VEL
LIN {X 0,Y 290.872,Z 1054.281,A -85,B 0,C 180,E1 -16639.207,E2 -16639.207} C_VEL
LIN {X 0,Y 290.45,Z 1060.967,A -85,B 0,C 180,E1 -16640.599,E2 -16640.599} C_VEL
LIN {X 0,Y 290.14,Z 1066.523,A -85,B 0,C 180,E1 -16641.993,E2 -16641.993} C_VEL
LIN {X 0,Y 289.938,Z 1071.198,A -85,B 0,C 180,E1 -16643.408,E2 -16643.408} C_VEL
LIN {X 0,Y 289.777,Z 1075.739,A -85,B 0,C 180,E1 -16645.13,E2 -16645.13} C_VEL
LIN {X 0,Y 289.616,Z 1078.637,A -85,B 0,C 180,E1 -16646.522,E2 -16646.522} C_VEL
LIN {X 0,Y 289.563,Z 1081.735,A -85,B 0,C 180,E1 -16648.609,E2 -16648.609} C_VEL
LIN {X 0,Y 289.593,Z 1083.084,A -85,B 0,C 180,E1 -16650,E2 -16650} C_VEL
LIN {X 0,Y 289.465,Z 1083.886,A -85,B 0,C 180,E1 -16651.391,E2 -16651.391} C_VEL
LIN {X 0,Y 289.503,Z 1084.108,A -85,B 0,C 180,E1 -16652.783,E2 -16652.783} C_VEL
LIN {X 0,Y 289.53,Z 1083.71,A -85,B 0,C 180,E1 -16654.176,E2 -16654.176} C_VEL
LIN {X 0,Y 289.635,Z 1082.607,A -85,B 0,C 180,E1 -16655.813,E2 -16655.813} C_VEL
LIN {X 0,Y 289.822,Z 1081.399,A -85,B 0,C 180,E1 -16656.964,E2 -16656.964} C_VEL
LIN {X 0,Y 290.439,Z 1078.191,A -85,B 0,C 180,E1 -16659.049,E2 -16659.049} C_VEL
LIN {X 0,Y 291.033,Z 1075.316,A -85,B 0,C 180,E1 -16660.434,E2 -16660.434} C_VEL
LIN {X 0,Y 292.296,Z 1069.763,A -85,B 0,C 180,E1 -16662.497,E2 -16662.497} C_VEL
LIN {X 0,Y 293.905,Z 1062.577,A -85,B 0,C 180,E1 -16664.541,E2 -16664.541} C_VEL
LIN {X 0,Y 295.53,Z 1054.85,A -85,B 0,C 180,E1 -16666.226,E2 -16666.226} C_VEL
LIN {X 0,Y 297.103,Z 1047.307,A -85,B 0,C 180,E1 -16667.554,E2 -16667.554} C_VEL
LIN {X 0,Y 298.879,Z 1038.261,A -85,B 0,C 180,E1 -16668.864,E2 -16668.864} C_VEL
LIN {X 0,Y 300.684,Z 1028.408,A -85,B 0,C 180,E1 -16669.989,E2 -16669.989} C_VEL
LIN {X 0,Y 302.436,Z 1017.388,A -85,B 0,C 180,E1 -16670.933,E2 -16670.933} C_VEL
LIN {X 0,Y 303.835,Z 1006.618,A -85,B 0,C 180,E1 -16671.632,E2 -16671.632} C_VEL
LIN {X 0,Y 305.362,Z 989.21,A -85,B 0,C 180,E1 -16672.39,E2 -16672.39} C_VEL
LIN {X 0,Y 307.142,Z 963.866,A -85,B 0,C 180,E1 -16673.426,E2 -16673.426} C_VEL
LIN {X 0,Y 306.341,Z 954.004,A -85,B 0,C 180,E1 -16674.081,E2 -16674.081} C_VEL
LIN {X 0,Y 304.124,Z 941.677,A -85,B 0,C 180,E1 -16675.156,E2 -16675.156} C_VEL
LIN {X 0,Y 301.993,Z 932.939,A -85,B 0,C 180,E1 -16676.069,E2 -16676.069} C_VEL
LIN {X 0,Y 300.859,Z 929.846,A -85,B 0,C 180,E1 -16676.484,E2 -16676.484} C_VEL
LIN {X 0,Y 299.047,Z 925.75,A -85,B 0,C 180,E1 -16677.134,E2 -16677.134} C_VEL
LIN {X 0,Y 296.91,Z 921.587,A -85,B 0,C 180,E1 -16677.874,E2 -16677.874} C_VEL
LIN {X 0,Y 296.67,Z 920.832,A -85,B 0,C 180,E1 -16678.032,E2 -16678.032} C_VEL
LIN {X 0,Y 295.665,Z 915.22,A -85,B 0,C 180,E1 -16681.161,E2 -16681.161} C_VEL
LIN {X 0,Y 294.64,Z 910.843,A -85,B 0,C 180,E1 -16684.092,E2 -16684.092} C_VEL
LIN {X 0,Y 293.772,Z 907.622,A -85,B 0,C 180,E1 -16686.732,E2 -16686.732} C_VEL
LIN {X 0,Y 292.801,Z 904.26,A -85,B 0,C 180,E1 -16690.396,E2 -16690.396} C_VEL
LIN {X 0,Y 292.191,Z 902.307,A -85,B 0,C 180,E1 -16693.815,E2 -16693.815} C_VEL
LIN {X 0,Y 292.036,Z 901.565,A -85,B 0,C 180,E1 -16696.217,E2 -16696.217} C_VEL
LIN {X 0,Y 291.989,Z 901.441,A -85,B 0,C 180,E1 -16699.469,E2 -16699.469} C_VEL
LIN {X 0,Y 292.273,Z 902.444,A -85,B 0,C 180,E1 -16703.048,E2 -16703.048} C_VEL
LIN {X 0,Y 292.59,Z 903.314,A -85,B 0,C 180,E1 -16704.797,E2 -16704.797} C_VEL
LIN {X 0,Y 293.191,Z 905.812,A -85,B 0,C 180,E1 -16708.174,E2 -16708.174} C_VEL
LIN {X 0,Y 294.005,Z 909.162,A -85,B 0,C 180,E1 -16711.44,E2 -16711.44} C_VEL
LIN {X 0,Y 296.112,Z 912.714,A -85,B 0,C 180,E1 -16712.239,E2 -16712.239} C_VEL
LIN {X 0,Y 297.448,Z 914.479,A -85,B 0,C 180,E1 -16712.687,E2 -16712.687} C_VEL
LIN {X 0,Y 300.737,Z 919.811,A -85,B 0,C 180,E1 -16713.769,E2 -16713.769} C_VEL
LIN {X 0,Y 304.32,Z 926.121,A -85,B 0,C 180,E1 -16714.882,E2 -16714.882} C_VEL
LIN {X 0,Y 308.396,Z 934.773,A -85,B 0,C 180,E1 -16716.126,E2 -16716.126} C_VEL
LIN {X 0,Y 308.907,Z 936.064,A -85,B 0,C 180,E1 -16716.281,E2 -16716.281} C_VEL
LIN {X 0,Y 304.912,Z 985.182,A -85,B 0,C 180,E1 -16718.293,E2 -16718.293} C_VEL
LIN {X 0,Y 303.635,Z 997.391,A -85,B 0,C 180,E1 -16719.065,E2 -16719.065} C_VEL
LIN {X 0,Y 302.257,Z 1007.549,A -85,B 0,C 180,E1 -16719.943,E2 -16719.943} C_VEL
LIN {X 0,Y 300.703,Z 1017.69,A -85,B 0,C 180,E1 -16721.078,E2 -16721.078} C_VEL
LIN {X 0,Y 298.81,Z 1027.716,A -85,B 0,C 180,E1 -16722.55,E2 -16722.55} C_VEL
LIN {X 0,Y 297.279,Z 1034.96,A -85,B 0,C 180,E1 -16723.873,E2 -16723.873} C_VEL
LIN {X 0,Y 295.903,Z 1041.026,A -85,B 0,C 180,E1 -16725.208,E2 -16725.208} C_VEL
LIN {X 0,Y 294.331,Z 1047.256,A -85,B 0,C 180,E1 -16726.89,E2 -16726.89} C_VEL
LIN {X 0,Y 292.84,Z 1053.012,A -85,B 0,C 180,E1 -16728.931,E2 -16728.931} C_VEL
LIN {X 0,Y 291.759,Z 1057.125,A -85,B 0,C 180,E1 -16730.976,E2 -16730.976} C_VEL
LIN {X 0,Y 290.736,Z 1060.044,A -85,B 0,C 180,E1 -16733.059,E2 -16733.059} C_VEL
LIN {X 0,Y 290.242,Z 1061.245,A -85,B 0,C 180,E1 -16734.442,E2 -16734.442} C_VEL
LIN {X 0,Y 289.96,Z 1061.928,A -85,B 0,C 180,E1 -16735.831,E2 -16735.831} C_VEL
LIN {X 0,Y 289.763,Z 1062.096,A -85,B 0,C 180,E1 -16737.22,E2 -16737.22} C_VEL
LIN {X 0,Y 289.593,Z 1061.653,A -85,B 0,C 180,E1 -16738.61,E2 -16738.61} C_VEL
LIN {X 0,Y 289.499,Z 1060.655,A -85,B 0,C 180,E1 -16740.001,E2 -16740.001} C_VEL
LIN {X 0,Y 289.519,Z 1058.213,A -85,B 0,C 180,E1 -16742.087,E2 -16742.087} C_VEL
LIN {X 0,Y 289.693,Z 1054.371,A -85,B 0,C 180,E1 -16744.174,E2 -16744.174} C_VEL
LIN {X 0,Y 289.834,Z 1049.998,A -85,B 0,C 180,E1 -16745.916,E2 -16745.916} C_VEL
LIN {X 0,Y 290.198,Z 1044.446,A -85,B 0,C 180,E1 -16747.655,E2 -16747.655} C_VEL
LIN {X 0,Y 290.503,Z 1039,A -85,B 0,C 180,E1 -16749.048,E2 -16749.048} C_VEL
LIN {X 0,Y 290.994,Z 1032.468,A -85,B 0,C 180,E1 -16750.437,E2 -16750.437} C_VEL
LIN {X 0,Y 291.627,Z 1023.518,A -85,B 0,C 180,E1 -16751.997,E2 -16751.997} C_VEL
LIN {X 0,Y 292.364,Z 1013.302,A -85,B 0,C 180,E1 -16753.379,E2 -16753.379} C_VEL
LIN {X 0,Y 293.017,Z 1003.619,A -85,B 0,C 180,E1 -16754.41,E2 -16754.41} C_VEL
LIN {X 0,Y 293.495,Z 994.342,A -85,B 0,C 180,E1 -16755.184,E2 -16755.184} C_VEL
LIN {X 0,Y 293.856,Z 982.361,A -85,B 0,C 180,E1 -16755.921,E2 -16755.921} C_VEL
LIN {X 0,Y 294.591,Z 959.608,A -85,B 0,C 180,E1 -16756.764,E2 -16756.764} C_VEL
LIN {X 0,Y 295.452,Z 926.661,A -85,B 0,C 180,E1 -16757.92,E2 -16757.92} C_VEL
LIN {X 0,Y 291.977,Z 902.55,A -85,B 0,C 180,E1 -16758.916,E2 -16758.916} C_VEL
LIN {X 0,Y 291.54,Z 898.975,A -85,B 0,C 180,E1 -16760.36,E2 -16760.36} C_VEL
LIN {X 0,Y 291.326,Z 899.005,A -85,B 0,C 180,E1 -16764.213,E2 -16764.213} C_VEL
LIN {X 0,Y 291.35,Z 899.007,A -85,B 0,C 180,E1 -16767.28,E2 -16767.28} C_VEL
LIN {X 0,Y 291.319,Z 899.005,A -85,B 0,C 180,E1 -16770.44,E2 -16770.44} C_VEL
LIN {X 0,Y 291.345,Z 899.007,A -85,B 0,C 180,E1 -16773.699,E2 -16773.699} C_VEL
LIN {X 0,Y 291.354,Z 899.004,A -85,B 0,C 180,E1 -16777.248,E2 -16777.248} C_VEL
LIN {X 0,Y 291.296,Z 899.012,A -85,B 0,C 180,E1 -16781.589,E2 -16781.589} C_VEL
LIN {X 0,Y 291.284,Z 899.012,A -85,B 0,C 180,E1 -16785.597,E2 -16785.597} C_VEL
LIN {X 0,Y 291.302,Z 899.007,A -85,B 0,C 180,E1 -16789.352,E2 -16789.352} C_VEL
LIN {X 0,Y 291.388,Z 898.999,A -85,B 0,C 180,E1 -16792.917,E2 -16792.917} C_VEL
LIN {X 0,Y 291.347,Z 899.006,A -85,B 0,C 180,E1 -16796.302,E2 -16796.302} C_VEL
LIN {X 0,Y 291.367,Z 899.002,A -85,B 0,C 180,E1 -16800.269,E2 -16800.269} C_VEL
LIN {X 0,Y 291.361,Z 899.002,A -85,B 0,C 180,E1 -16804.267,E2 -16804.267} C_VEL
LIN {X 0,Y 291.366,Z 899.002,A -85,B 0,C 180,E1 -16807.298,E2 -16807.298} C_VEL
LIN {X 0,Y 291.392,Z 898.997,A -85,B 0,C 180,E1 -16810.266,E2 -16810.266} C_VEL
LIN {X 0,Y 291.502,Z 898.984,A -85,B 0,C 180,E1 -16814.666,E2 -16814.666} C_VEL
LIN {X 0,Y 291.531,Z 898.98,A -85,B 0,C 180,E1 -16818.881,E2 -16818.881} C_VEL
LIN {X 0,Y 291.656,Z 898.969,A -85,B 0,C 180,E1 -16821.687,E2 -16821.687} C_VEL
LIN {X 0,Y 291.597,Z 898.971,A -85,B 0,C 180,E1 -16824.468,E2 -16824.468} C_VEL
LIN {X 0,Y 291.87,Z 898.938,A -85,B 0,C 180,E1 -16828.62,E2 -16828.62} C_VEL
LIN {X 0,Y 291.87,Z 898.938,A -85,B 0,C 180,E1 -16831.38,E2 -16831.38} C_VEL
LIN {X 0,Y 291.69,Z 898.961,A -85,B 0,C 180,E1 -16836.92,E2 -16836.92} C_VEL
LIN {X 0,Y 291.572,Z 898.975,A -85,B 0,C 180,E1 -16839.714,E2 -16839.714} C_VEL
LIN {X 0,Y 291.48,Z 898.985,A -85,B 0,C 180,E1 -16843.953,E2 -16843.953} C_VEL
LIN {X 0,Y 291.382,Z 899,A -85,B 0,C 180,E1 -16848.274,E2 -16848.274} C_VEL
LIN {X 0,Y 291.346,Z 899.005,A -85,B 0,C 180,E1 -16851.213,E2 -16851.213} C_VEL
LIN {X 0,Y 291.33,Z 899.004,A -85,B 0,C 180,E1 -16854.212,E2 -16854.212} C_VEL
LIN {X 0,Y 291.354,Z 899.007,A -85,B 0,C 180,E1 -16857.279,E2 -16857.279} C_VEL
LIN {X 0,Y 291.322,Z 899.005,A -85,B 0,C 180,E1 -16860.439,E2 -16860.439} C_VEL
LIN {X 0,Y 291.348,Z 899.006,A -85,B 0,C 180,E1 -16863.698,E2 -16863.698} C_VEL
LIN {X 0,Y 291.356,Z 899.004,A -85,B 0,C 180,E1 -16867.247,E2 -16867.247} C_VEL
LIN {X 0,Y 291.303,Z 899.007,A -85,B 0,C 180,E1 -16870.648,E2 -16870.648} C_VEL
LIN {X 0,Y 291.286,Z 899.012,A -85,B 0,C 180,E1 -16874.403,E2 -16874.403} C_VEL
LIN {X 0,Y 291.298,Z 899.011,A -85,B 0,C 180,E1 -16878.411,E2 -16878.411} C_VEL
LIN {X 0,Y 291.336,Z 899.003,A -85,B 0,C 180,E1 -16881.155,E2 -16881.155} C_VEL
LIN {X 0,Y 291.359,Z 899.005,A -85,B 0,C 180,E1 -16884.625,E2 -16884.625} C_VEL
LIN {X 0,Y 291.37,Z 899,A -85,B 0,C 180,E1 -16887.95,E2 -16887.95} C_VEL
LIN {X 0,Y 291.345,Z 899.004,A -85,B 0,C 180,E1 -16891.153,E2 -16891.153} C_VEL
LIN {X 0,Y 291.345,Z 899.004,A -85,B 0,C 180,E1 -16894.264,E2 -16894.264} C_VEL
LIN {X 0,Y 291.352,Z 899.004,A -85,B 0,C 180,E1 -16897.296,E2 -16897.296} C_VEL
LIN {X 0,Y 291.387,Z 898.997,A -85,B 0,C 180,E1 -16900.264,E2 -16900.264} C_VEL
LIN {X 0,Y 291.455,Z 898.99,A -85,B 0,C 180,E1 -16904.698,E2 -16904.698} C_VEL
LIN {X 0,Y 291.528,Z 898.98,A -85,B 0,C 180,E1 -16908.88,E2 -16908.88} C_VEL
LIN {X 0,Y 291.655,Z 898.97,A -85,B 0,C 180,E1 -16911.686,E2 -16911.686} C_VEL
LIN {X 0,Y 291.595,Z 898.972,A -85,B 0,C 180,E1 -16914.467,E2 -16914.467} C_VEL
LIN {X 0,Y 291.867,Z 898.938,A -85,B 0,C 180,E1 -16918.62,E2 -16918.62} C_VEL
LIN {X 0,Y 291.867,Z 898.938,A -85,B 0,C 180,E1 -16921.379,E2 -16921.379} C_VEL
LIN {X 0,Y 291.64,Z 898.966,A -85,B 0,C 180,E1 -16923.236,E2 -16923.236} C_VEL
LIN {X 0,Y 290.847,Z 899.068,A -85,B 0,C 180,E1 -16924.389,E2 -16924.389} C_VEL
LIN {X 0,Y 288.041,Z 899.419,A -85,B 0,C 180,E1 -16926.27,E2 -16926.27} C_VEL
LIN {X 0,Y 284.919,Z 899.807,A -85,B 0,C 180,E1 -16928.579,E2 -16928.579} C_VEL
LIN {X 0,Y 284.562,Z 899.848,A -85,B 0,C 180,E1 -16929.376,E2 -16929.376} C_VEL
LIN {X 0,Y 284.455,Z 899.864,A -85,B 0,C 180,E1 -16932.847,E2 -16932.847} C_VEL
LIN {X 0,Y 284.393,Z 899.868,A -85,B 0,C 180,E1 -16935.773,E2 -16935.773} C_VEL
LIN {X 0,Y 284.323,Z 899.878,A -85,B 0,C 180,E1 -16940.246,E2 -16940.246} C_VEL
LIN {X 0,Y 284.293,Z 899.881,A -85,B 0,C 180,E1 -16943.839,E2 -16943.839} C_VEL
LIN {X 0,Y 284.281,Z 899.883,A -85,B 0,C 180,E1 -16948.015,E2 -16948.015} C_VEL
LIN {X 0,Y 284.285,Z 899.887,A -85,B 0,C 180,E1 -16951.275,E2 -16951.275} C_VEL
LIN {X 0,Y 284.336,Z 899.878,A -85,B 0,C 180,E1 -16955.346,E2 -16955.346} C_VEL
LIN {X 0,Y 284.295,Z 899.883,A -85,B 0,C 180,E1 -16958.171,E2 -16958.171} C_VEL
LIN {X 0,Y 284.236,Z 899.891,A -85,B 0,C 180,E1 -16962.116,E2 -16962.116} C_VEL
LIN {X 0,Y 284.237,Z 899.893,A -85,B 0,C 180,E1 -16966.185,E2 -16966.185} C_VEL
LIN {X 0,Y 284.282,Z 899.886,A -85,B 0,C 180,E1 -16970.029,E2 -16970.029} C_VEL
LIN {X 0,Y 284.317,Z 899.877,A -85,B 0,C 180,E1 -16973.611,E2 -16973.611} C_VEL
LIN {X 0,Y 284.305,Z 899.881,A -85,B 0,C 180,E1 -16977.19,E2 -16977.19} C_VEL
LIN {X 0,Y 284.422,Z 899.989,A -85,B 0,C 180,E1 -16981.898,E2 -16981.898} C_VEL
LIN {X 0,Y 286.389,Z 910.66,A -85,B 0,C 180,E1 -16985.729,E2 -16985.729} C_VEL
LIN {X 0,Y 286.196,Z 915.084,A -85,B 0,C 180,E1 -16987.246,E2 -16987.246} C_VEL
LIN {X 0,Y 284.92,Z 925.542,A -85,B 0,C 180,E1 -16990.783,E2 -16990.783} C_VEL
LIN {X 0,Y 286.477,Z 946.198,A -85,B 0,C 180,E1 -16991.63,E2 -16991.63} C_VEL
LIN {X 0,Y 288.07,Z 961.918,A -85,B 0,C 180,E1 -16992.262,E2 -16992.262} C_VEL
LIN {X 0,Y 286.915,Z 1004.392,A -85,B 0,C 180,E1 -16993.867,E2 -16993.867} C_VEL
LIN {X 0,Y 286.287,Z 1015.562,A -85,B 0,C 180,E1 -16994.516,E2 -16994.516} C_VEL
LIN {X 0,Y 285.798,Z 1026.106,A -85,B 0,C 180,E1 -16995.4,E2 -16995.4} C_VEL
LIN {X 0,Y 285.198,Z 1034.367,A -85,B 0,C 180,E1 -16996.279,E2 -16996.279} C_VEL
LIN {X 0,Y 284.634,Z 1042.498,A -85,B 0,C 180,E1 -16997.341,E2 -16997.341} C_VEL
LIN {X 0,Y 284.091,Z 1050.323,A -85,B 0,C 180,E1 -16998.585,E2 -16998.585} C_VEL
LIN {X 0,Y 283.443,Z 1059.385,A -85,B 0,C 180,E1 -17000.365,E2 -17000.365} C_VEL
LIN {X 0,Y 283.05,Z 1066.388,A -85,B 0,C 180,E1 -17002.151,E2 -17002.151} C_VEL
LIN {X 0,Y 282.804,Z 1071.42,A -85,B 0,C 180,E1 -17003.741,E2 -17003.741} C_VEL
LIN {X 0,Y 282.662,Z 1076.335,A -85,B 0,C 180,E1 -17005.722,E2 -17005.722} C_VEL
LIN {X 0,Y 282.459,Z 1080.182,A -85,B 0,C 180,E1 -17007.861,E2 -17007.861} C_VEL
LIN {X 0,Y 282.51,Z 1082.558,A -85,B 0,C 180,E1 -17010,E2 -17010} C_VEL
LIN {X 0,Y 282.387,Z 1083.447,A -85,B 0,C 180,E1 -17011.426,E2 -17011.426} C_VEL
LIN {X 0,Y 282.431,Z 1083.719,A -85,B 0,C 180,E1 -17012.852,E2 -17012.852} C_VEL
LIN {X 0,Y 282.435,Z 1083.465,A -85,B 0,C 180,E1 -17014.281,E2 -17014.281} C_VEL
LIN {X 0,Y 282.52,Z 1082.71,A -85,B 0,C 180,E1 -17015.71,E2 -17015.71} C_VEL
LIN {X 0,Y 282.768,Z 1081.446,A -85,B 0,C 180,E1 -17017.138,E2 -17017.138} C_VEL
LIN {X 0,Y 283.427,Z 1078.397,A -85,B 0,C 180,E1 -17019.275,E2 -17019.275} C_VEL
LIN {X 0,Y 284.485,Z 1074.077,A -85,B 0,C 180,E1 -17021.398,E2 -17021.398} C_VEL
LIN {X 0,Y 285.665,Z 1069.343,A -85,B 0,C 180,E1 -17023.154,E2 -17023.154} C_VEL
LIN {X 0,Y 287.373,Z 1062.12,A -85,B 0,C 180,E1 -17025.242,E2 -17025.242} C_VEL
LIN {X 0,Y 289.197,Z 1054.442,A -85,B 0,C 180,E1 -17026.955,E2 -17026.955} C_VEL
LIN {X 0,Y 290.942,Z 1046.977,A -85,B 0,C 180,E1 -17028.302,E2 -17028.302} C_VEL
LIN {X 0,Y 292.85,Z 1037.93,A -85,B 0,C 180,E1 -17029.632,E2 -17029.632} C_VEL
LIN {X 0,Y 294.774,Z 1028.076,A -85,B 0,C 180,E1 -17030.772,E2 -17030.772} C_VEL
LIN {X 0,Y 296.659,Z 1017.231,A -85,B 0,C 180,E1 -17031.726,E2 -17031.726} C_VEL
LIN {X 0,Y 298.329,Z 1005.315,A -85,B 0,C 180,E1 -17032.518,E2 -17032.518} C_VEL
LIN {X 0,Y 299.959,Z 987.307,A -85,B 0,C 180,E1 -17033.31,E2 -17033.31} C_VEL
LIN {X 0,Y 301.67,Z 964.251,A -85,B 0,C 180,E1 -17034.289,E2 -17034.289} C_VEL
LIN {X 0,Y 300.839,Z 954.897,A -85,B 0,C 180,E1 -17034.982,E2 -17034.982} C_VEL
LIN {X 0,Y 298.714,Z 942.787,A -85,B 0,C 180,E1 -17036.103,E2 -17036.103} C_VEL
LIN {X 0,Y 296.815,Z 934.992,A -85,B 0,C 180,E1 -17037.008,E2 -17037.008} C_VEL
LIN {X 0,Y 294.62,Z 930.303,A -85,B 0,C 180,E1 -17037.803,E2 -17037.803} C_VEL
LIN {X 0,Y 292.263,Z 925.523,A -85,B 0,C 180,E1 -17038.724,E2 -17038.724} C_VEL
LIN {X 0,Y 289.786,Z 920.987,A -85,B 0,C 180,E1 -17039.701,E2 -17039.701} C_VEL
LIN {X 0,Y 289.553,Z 920.234,A -85,B 0,C 180,E1 -17039.84,E2 -17039.84} C_VEL
LIN {X 0,Y 288.728,Z 916.188,A -85,B 0,C 180,E1 -17042.378,E2 -17042.378} C_VEL
LIN {X 0,Y 287.656,Z 911.56,A -85,B 0,C 180,E1 -17045.899,E2 -17045.899} C_VEL
LIN {X 0,Y 286.631,Z 908.012,A -85,B 0,C 180,E1 -17049.606,E2 -17049.606} C_VEL
LIN {X 0,Y 286.057,Z 906.099,A -85,B 0,C 180,E1 -17052.52,E2 -17052.52} C_VEL
LIN {X 0,Y 285.677,Z 904.732,A -85,B 0,C 180,E1 -17056.463,E2 -17056.463} C_VEL
LIN {X 0,Y 285.705,Z 904.73,A -85,B 0,C 180,E1 -17060.241,E2 -17060.241} C_VEL
LIN {X 0,Y 286.06,Z 906.073,A -85,B 0,C 180,E1 -17064.169,E2 -17064.169} C_VEL
LIN {X 0,Y 286.554,Z 908.108,A -85,B 0,C 180,E1 -17067.346,E2 -17067.346} C_VEL
LIN {X 0,Y 287.094,Z 910.162,A -85,B 0,C 180,E1 -17069.531,E2 -17069.531} C_VEL
LIN {X 0,Y 289.388,Z 913.741,A -85,B 0,C 180,E1 -17070.532,E2 -17070.532} C_VEL
LIN {X 0,Y 290.842,Z 915.657,A -85,B 0,C 180,E1 -17071.1,E2 -17071.1} C_VEL
LIN {X 0,Y 293.96,Z 920.434,A -85,B 0,C 180,E1 -17072.267,E2 -17072.267} C_VEL
LIN {X 0,Y 297.289,Z 925.913,A -85,B 0,C 180,E1 -17073.424,E2 -17073.424} C_VEL
LIN {X 0,Y 301.58,Z 934.195,A -85,B 0,C 180,E1 -17074.848,E2 -17074.848} C_VEL
LIN {X 0,Y 303.503,Z 938.557,A -85,B 0,C 180,E1 -17075.47,E2 -17075.47} C_VEL
LIN {X 0,Y 299.33,Z 985.971,A -85,B 0,C 180,E1 -17077.481,E2 -17077.481} C_VEL
LIN {X 0,Y 298.081,Z 997.136,A -85,B 0,C 180,E1 -17078.202,E2 -17078.202} C_VEL
LIN {X 0,Y 296.44,Z 1008.089,A -85,B 0,C 180,E1 -17079.169,E2 -17079.169} C_VEL
LIN {X 0,Y 294.739,Z 1018.08,A -85,B 0,C 180,E1 -17080.318,E2 -17080.318} C_VEL
LIN {X 0,Y 292.72,Z 1028.125,A -85,B 0,C 180,E1 -17081.813,E2 -17081.813} C_VEL
LIN {X 0,Y 291.07,Z 1035.362,A -85,B 0,C 180,E1 -17083.158,E2 -17083.158} C_VEL
LIN {X 0,Y 289.592,Z 1041.366,A -85,B 0,C 180,E1 -17084.517,E2 -17084.517} C_VEL
LIN {X 0,Y 287.895,Z 1047.541,A -85,B 0,C 180,E1 -17086.231,E2 -17086.231} C_VEL
LIN {X 0,Y 286.454,Z 1052.514,A -85,B 0,C 180,E1 -17087.964,E2 -17087.964} C_VEL
LIN {X 0,Y 285.14,Z 1056.934,A -85,B 0,C 180,E1 -17090.066,E2 -17090.066} C_VEL
LIN {X 0,Y 284.44,Z 1059.161,A -85,B 0,C 180,E1 -17091.475,E2 -17091.475} C_VEL
LIN {X 0,Y 283.737,Z 1060.76,A -85,B 0,C 180,E1 -17092.886,E2 -17092.886} C_VEL
LIN {X 0,Y 283.214,Z 1061.796,A -85,B 0,C 180,E1 -17094.304,E2 -17094.304} C_VEL
LIN {X 0,Y 282.902,Z 1062.328,A -85,B 0,C 180,E1 -17095.727,E2 -17095.727} C_VEL
LIN {X 0,Y 282.689,Z 1062.358,A -85,B 0,C 180,E1 -17097.151,E2 -17097.151} C_VEL
LIN {X 0,Y 282.512,Z 1061.855,A -85,B 0,C 180,E1 -17098.575,E2 -17098.575} C_VEL
LIN {X 0,Y 282.416,Z 1060.737,A -85,B 0,C 180,E1 -17100.001,E2 -17100.001} C_VEL
LIN {X 0,Y 282.446,Z 1058.091,A -85,B 0,C 180,E1 -17102.14,E2 -17102.14} C_VEL
LIN {X 0,Y 282.614,Z 1054.003,A -85,B 0,C 180,E1 -17104.279,E2 -17104.279} C_VEL
LIN {X 0,Y 282.806,Z 1048.886,A -85,B 0,C 180,E1 -17106.26,E2 -17106.26} C_VEL
LIN {X 0,Y 283.251,Z 1042.442,A -85,B 0,C 180,E1 -17108.203,E2 -17108.203} C_VEL
LIN {X 0,Y 283.713,Z 1034.806,A -85,B 0,C 180,E1 -17109.986,E2 -17109.986} C_VEL
LIN {X 0,Y 284.394,Z 1026.234,A -85,B 0,C 180,E1 -17111.584,E2 -17111.584} C_VEL
LIN {X 0,Y 285.042,Z 1016.819,A -85,B 0,C 180,E1 -17113.003,E2 -17113.003} C_VEL
LIN {X 0,Y 285.717,Z 1006.187,A -85,B 0,C 180,E1 -17114.24,E2 -17114.24} C_VEL
LIN {X 0,Y 286.289,Z 996.413,A -85,B 0,C 180,E1 -17115.12,E2 -17115.12} C_VEL
LIN {X 0,Y 286.579,Z 986.755,A -85,B 0,C 180,E1 -17115.788,E2 -17115.788} C_VEL
LIN {X 0,Y 287.13,Z 973.92,A -85,B 0,C 180,E1 -17116.395,E2 -17116.395} C_VEL
LIN {X 0,Y 288.39,Z 927.025,A -85,B 0,C 180,E1 -17118.117,E2 -17118.117} C_VEL
LIN {X 0,Y 284.89,Z 902.877,A -85,B 0,C 180,E1 -17119.126,E2 -17119.126} C_VEL
LIN {X 0,Y 284.495,Z 899.847,A -85,B 0,C 180,E1 -17120.423,E2 -17120.423} C_VEL
LIN {X 0,Y 284.284,Z 899.886,A -85,B 0,C 180,E1 -17124.852,E2 -17124.852} C_VEL
LIN {X 0,Y 284.281,Z 899.882,A -85,B 0,C 180,E1 -17128.017,E2 -17128.017} C_VEL
LIN {X 0,Y 284.286,Z 899.885,A -85,B 0,C 180,E1 -17131.276,E2 -17131.276} C_VEL
LIN {X 0,Y 284.338,Z 899.879,A -85,B 0,C 180,E1 -17135.347,E2 -17135.347} C_VEL
LIN {X 0,Y 284.265,Z 899.885,A -85,B 0,C 180,E1 -17138.178,E2 -17138.178} C_VEL
LIN {X 0,Y 284.238,Z 899.891,A -85,B 0,C 180,E1 -17142.118,E2 -17142.118} C_VEL
LIN {X 0,Y 284.24,Z 899.892,A -85,B 0,C 180,E1 -17146.186,E2 -17146.186} C_VEL
LIN {X 0,Y 284.286,Z 899.885,A -85,B 0,C 180,E1 -17150.03,E2 -17150.03} C_VEL
LIN {X 0,Y 284.321,Z 899.878,A -85,B 0,C 180,E1 -17153.613,E2 -17153.613} C_VEL
LIN {X 0,Y 284.309,Z 899.878,A -85,B 0,C 180,E1 -17157.191,E2 -17157.191} C_VEL
LIN {X 0,Y 284.339,Z 899.878,A -85,B 0,C 180,E1 -17160.374,E2 -17160.374} C_VEL
LIN {X 0,Y 284.308,Z 899.88,A -85,B 0,C 180,E1 -17163.58,E2 -17163.58} C_VEL
LIN {X 0,Y 284.33,Z 899.879,A -85,B 0,C 180,E1 -17166.704,E2 -17166.704} C_VEL
LIN {X 0,Y 284.33,Z 899.882,A -85,B 0,C 180,E1 -17171.257,E2 -17171.257} C_VEL
LIN {X 0,Y 284.466,Z 899.861,A -85,B 0,C 180,E1 -17175.697,E2 -17175.697} C_VEL
LIN {X 0,Y 284.518,Z 899.855,A -85,B 0,C 180,E1 -17180.043,E2 -17180.043} C_VEL
LIN {X 0,Y 284.646,Z 899.837,A -85,B 0,C 180,E1 -17182.909,E2 -17182.909} C_VEL
LIN {X 0,Y 284.837,Z 899.814,A -85,B 0,C 180,E1 -17188.586,E2 -17188.586} C_VEL
LIN {X 0,Y 284.836,Z 899.814,A -85,B 0,C 180,E1 -17191.414,E2 -17191.414} C_VEL
LIN {X 0,Y 284.646,Z 899.837,A -85,B 0,C 180,E1 -17197.092,E2 -17197.092} C_VEL
LIN {X 0,Y 284.518,Z 899.855,A -85,B 0,C 180,E1 -17199.957,E2 -17199.957} C_VEL
LIN {X 0,Y 284.413,Z 899.867,A -85,B 0,C 180,E1 -17204.307,E2 -17204.307} C_VEL
LIN {X 0,Y 284.346,Z 899.876,A -85,B 0,C 180,E1 -17207.254,E2 -17207.254} C_VEL
LIN {X 0,Y 284.327,Z 899.878,A -85,B 0,C 180,E1 -17210.246,E2 -17210.246} C_VEL
LIN {X 0,Y 284.297,Z 899.88,A -85,B 0,C 180,E1 -17213.84,E2 -17213.84} C_VEL
LIN {X 0,Y 284.285,Z 899.883,A -85,B 0,C 180,E1 -17218.016,E2 -17218.016} C_VEL
LIN {X 0,Y 284.289,Z 899.886,A -85,B 0,C 180,E1 -17221.276,E2 -17221.276} C_VEL
LIN {X 0,Y 284.341,Z 899.879,A -85,B 0,C 180,E1 -17225.346,E2 -17225.346} C_VEL
LIN {X 0,Y 284.299,Z 899.882,A -85,B 0,C 180,E1 -17228.172,E2 -17228.172} C_VEL
LIN {X 0,Y 284.24,Z 899.89,A -85,B 0,C 180,E1 -17232.117,E2 -17232.117} C_VEL
LIN {X 0,Y 284.242,Z 899.892,A -85,B 0,C 180,E1 -17236.185,E2 -17236.185} C_VEL
LIN {X 0,Y 284.287,Z 899.885,A -85,B 0,C 180,E1 -17240.029,E2 -17240.029} C_VEL
LIN {X 0,Y 284.322,Z 899.878,A -85,B 0,C 180,E1 -17243.612,E2 -17243.612} C_VEL
LIN {X 0,Y 284.31,Z 899.88,A -85,B 0,C 180,E1 -17247.19,E2 -17247.19} C_VEL
LIN {X 0,Y 284.34,Z 899.877,A -85,B 0,C 180,E1 -17250.373,E2 -17250.373} C_VEL
LIN {X 0,Y 284.3,Z 899.881,A -85,B 0,C 180,E1 -17253.578,E2 -17253.578} C_VEL
LIN {X 0,Y 284.31,Z 899.882,A -85,B 0,C 180,E1 -17256.701,E2 -17256.701} C_VEL
LIN {X 0,Y 284.337,Z 899.875,A -85,B 0,C 180,E1 -17259.928,E2 -17259.928} C_VEL
LIN {X 0,Y 284.423,Z 899.865,A -85,B 0,C 180,E1 -17264.512,E2 -17264.512} C_VEL
LIN {X 0,Y 284.464,Z 899.858,A -85,B 0,C 180,E1 -17268.6,E2 -17268.6} C_VEL
LIN {X 0,Y 284.612,Z 899.846,A -85,B 0,C 180,E1 -17271.479,E2 -17271.479} C_VEL
LIN {X 0,Y 284.566,Z 899.848,A -85,B 0,C 180,E1 -17274.33,E2 -17274.33} C_VEL
LIN {X 0,Y 284.834,Z 899.814,A -85,B 0,C 180,E1 -17278.585,E2 -17278.585} C_VEL
LIN {X 0,Y 284.834,Z 899.815,A -85,B 0,C 180,E1 -17281.413,E2 -17281.413} C_VEL
LIN {X 0,Y 284.643,Z 899.837,A -85,B 0,C 180,E1 -17287.091,E2 -17287.091} C_VEL
LIN {X 0,Y 284.562,Z 899.848,A -85,B 0,C 180,E1 -17289.376,E2 -17289.376} C_VEL
LIN {X 0,Y 283.797,Z 899.948,A -85,B 0,C 180,E1 -17290.556,E2 -17290.556} C_VEL
LIN {X 0,Y 280.858,Z 900.314,A -85,B 0,C 180,E1 -17292.477,E2 -17292.477} C_VEL
LIN {X 0,Y 278.437,Z 900.613,A -85,B 0,C 180,E1 -17294.038,E2 -17294.038} C_VEL
LIN {X 0,Y 277.435,Z 900.736,A -85,B 0,C 180,E1 -17295.248,E2 -17295.248} C_VEL
LIN {X 0,Y 277.37,Z 900.742,A -85,B 0,C 180,E1 -17295.658,E2 -17295.658} C_VEL
LIN {X 0,Y 277.273,Z 900.757,A -85,B 0,C 180,E1 -17300.308,E2 -17300.308} C_VEL
LIN {X 0,Y 277.237,Z 900.759,A -85,B 0,C 180,E1 -17304.131,E2 -17304.131} C_VEL
LIN {X 0,Y 277.267,Z 900.76,A -85,B 0,C 180,E1 -17307.481,E2 -17307.481} C_VEL
LIN {X 0,Y 277.248,Z 900.759,A -85,B 0,C 180,E1 -17310.472,E2 -17310.472} C_VEL
LIN {X 0,Y 277.246,Z 900.76,A -85,B 0,C 180,E1 -17313.895,E2 -17313.895} C_VEL
LIN {X 0,Y 277.25,Z 900.762,A -85,B 0,C 180,E1 -17317.471,E2 -17317.471} C_VEL
LIN {X 0,Y 277.183,Z 900.768,A -85,B 0,C 180,E1 -17321.241,E2 -17321.241} C_VEL
LIN {X 0,Y 277.173,Z 900.767,A -85,B 0,C 180,E1 -17325.232,E2 -17325.232} C_VEL
LIN {X 0,Y 277.183,Z 900.768,A -85,B 0,C 180,E1 -17328.758,E2 -17328.758} C_VEL
LIN {X 0,Y 277.25,Z 900.761,A -85,B 0,C 180,E1 -17332.527,E2 -17332.527} C_VEL
LIN {X 0,Y 277.245,Z 900.761,A -85,B 0,C 180,E1 -17336.104,E2 -17336.104} C_VEL
LIN {X 0,Y 277.261,Z 900.757,A -85,B 0,C 180,E1 -17339.538,E2 -17339.538} C_VEL
LIN {X 0,Y 277.405,Z 900.932,A -85,B 0,C 180,E1 -17341.864,E2 -17341.864} C_VEL
LIN {X 0,Y 279.326,Z 911.288,A -85,B 0,C 180,E1 -17345.68,E2 -17345.68} C_VEL
LIN {X 0,Y 279.16,Z 915.135,A -85,B 0,C 180,E1 -17347.031,E2 -17347.031} C_VEL
LIN {X 0,Y 277.9,Z 925.304,A -85,B 0,C 180,E1 -17350.566,E2 -17350.566} C_VEL
LIN {X 0,Y 279.124,Z 943.532,A -85,B 0,C 180,E1 -17351.343,E2 -17351.343} C_VEL
LIN {X 0,Y 280.994,Z 962.575,A -85,B 0,C 180,E1 -17352.135,E2 -17352.135} C_VEL
LIN {X 0,Y 279.853,Z 1004.219,A -85,B 0,C 180,E1 -17353.776,E2 -17353.776} C_VEL
LIN {X 0,Y 279.159,Z 1015.874,A -85,B 0,C 180,E1 -17354.485,E2 -17354.485} C_VEL
LIN {X 0,Y 278.671,Z 1026.256,A -85,B 0,C 180,E1 -17355.392,E2 -17355.392} C_VEL
LIN {X 0,Y 277.976,Z 1035.9,A -85,B 0,C 180,E1 -17356.475,E2 -17356.475} C_VEL
LIN {X 0,Y 277.239,Z 1046.123,A -85,B 0,C 180,E1 -17357.928,E2 -17357.928} C_VEL
LIN {X 0,Y 276.675,Z 1054.139,A -85,B 0,C 180,E1 -17359.387,E2 -17359.387} C_VEL
LIN {X 0,Y 276.255,Z 1060.758,A -85,B 0,C 180,E1 -17360.851,E2 -17360.851} C_VEL
LIN {X 0,Y 275.921,Z 1067.481,A -85,B 0,C 180,E1 -17362.683,E2 -17362.683} C_VEL
LIN {X 0,Y 275.704,Z 1071.795,A -85,B 0,C 180,E1 -17364.147,E2 -17364.147} C_VEL
LIN {X 0,Y 275.61,Z 1075.325,A -85,B 0,C 180,E1 -17365.612,E2 -17365.612} C_VEL
LIN {X 0,Y 275.433,Z 1078.146,A -85,B 0,C 180,E1 -17367.075,E2 -17367.075} C_VEL
LIN {X 0,Y 275.41,Z 1080.361,A -85,B 0,C 180,E1 -17368.537,E2 -17368.537} C_VEL
LIN {X 0,Y 275.432,Z 1081.963,A -85,B 0,C 180,E1 -17370,E2 -17370} C_VEL
LIN {X 0,Y 275.31,Z 1082.907,A -85,B 0,C 180,E1 -17371.463,E2 -17371.463} C_VEL
LIN {X 0,Y 275.361,Z 1083.321,A -85,B 0,C 180,E1 -17372.926,E2 -17372.926} C_VEL
LIN {X 0,Y 275.344,Z 1083.219,A -85,B 0,C 180,E1 -17374.391,E2 -17374.391} C_VEL
LIN {X 0,Y 275.448,Z 1082.62,A -85,B 0,C 180,E1 -17375.857,E2 -17375.857} C_VEL
LIN {X 0,Y 275.716,Z 1081.454,A -85,B 0,C 180,E1 -17377.322,E2 -17377.322} C_VEL
LIN {X 0,Y 276.431,Z 1078.663,A -85,B 0,C 180,E1 -17379.512,E2 -17379.512} C_VEL
LIN {X 0,Y 277.561,Z 1074.507,A -85,B 0,C 180,E1 -17381.687,E2 -17381.687} C_VEL
LIN {X 0,Y 279.1,Z 1068.975,A -85,B 0,C 180,E1 -17383.84,E2 -17383.84} C_VEL
LIN {X 0,Y 280.612,Z 1063.141,A -85,B 0,C 180,E1 -17385.619,E2 -17385.619} C_VEL
LIN {X 0,Y 282.545,Z 1055.878,A -85,B 0,C 180,E1 -17387.367,E2 -17387.367} C_VEL
LIN {X 0,Y 284.589,Z 1047.707,A -85,B 0,C 180,E1 -17388.912,E2 -17388.912} C_VEL
LIN {X 0,Y 286.344,Z 1040.179,A -85,B 0,C 180,E1 -17390.097,E2 -17390.097} C_VEL
LIN {X 0,Y 287.994,Z 1032.494,A -85,B 0,C 180,E1 -17391.097,E2 -17391.097} C_VEL
LIN {X 0,Y 289.935,Z 1023.091,A -85,B 0,C 180,E1 -17392.069,E2 -17392.069} C_VEL
LIN {X 0,Y 291.996,Z 1010.992,A -85,B 0,C 180,E1 -17393.024,E2 -17393.024} C_VEL
LIN {X 0,Y 293.486,Z 999.03,A -85,B 0,C 180,E1 -17393.694,E2 -17393.694} C_VEL
LIN {X 0,Y 296.387,Z 965.716,A -85,B 0,C 180,E1 -17395.155,E2 -17395.155} C_VEL
LIN {X 0,Y 295.587,Z 956.543,A -85,B 0,C 180,E1 -17395.861,E2 -17395.861} C_VEL
LIN {X 0,Y 293.362,Z 943.051,A -85,B 0,C 180,E1 -17397.22,E2 -17397.22} C_VEL
LIN {X 0,Y 291.898,Z 938.249,A -85,B 0,C 180,E1 -17397.882,E2 -17397.882} C_VEL
LIN {X 0,Y 290.273,Z 934.609,A -85,B 0,C 180,E1 -17398.549,E2 -17398.549} C_VEL
LIN {X 0,Y 288.331,Z 930.593,A -85,B 0,C 180,E1 -17399.348,E2 -17399.348} C_VEL
LIN {X 0,Y 285.63,Z 925.367,A -85,B 0,C 180,E1 -17400.551,E2 -17400.551} C_VEL
LIN {X 0,Y 282.94,Z 920.899,A -85,B 0,C 180,E1 -17401.796,E2 -17401.796} C_VEL
LIN {X 0,Y 282.324,Z 919.382,A -85,B 0,C 180,E1 -17402.181,E2 -17402.181} C_VEL
LIN {X 0,Y 281.462,Z 915.591,A -85,B 0,C 180,E1 -17405.051,E2 -17405.051} C_VEL
LIN {X 0,Y 280.415,Z 911.82,A -85,B 0,C 180,E1 -17408.797,E2 -17408.797} C_VEL
LIN {X 0,Y 279.955,Z 910.073,A -85,B 0,C 180,E1 -17411.139,E2 -17411.139} C_VEL
LIN {X 0,Y 279.39,Z 908.228,A -85,B 0,C 180,E1 -17415.225,E2 -17415.225} C_VEL
LIN {X 0,Y 279.323,Z 907.831,A -85,B 0,C 180,E1 -17417.208,E2 -17417.208} C_VEL
LIN {X 0,Y 279.3,Z 907.798,A -85,B 0,C 180,E1 -17419.139,E2 -17419.139} C_VEL
LIN {X 0,Y 279.477,Z 908.646,A -85,B 0,C 180,E1 -17422.878,E2 -17422.878} C_VEL
LIN {X 0,Y 280.024,Z 910.521,A -85,B 0,C 180,E1 -17426.486,E2 -17426.486} C_VEL
LIN {X 0,Y 280.175,Z 911.146,A -85,B 0,C 180,E1 -17427.149,E2 -17427.149} C_VEL
LIN {X 0,Y 282.499,Z 914.736,A -85,B 0,C 180,E1 -17428.398,E2 -17428.398} C_VEL
LIN {X 0,Y 284.102,Z 916.476,A -85,B 0,C 180,E1 -17429.143,E2 -17429.143} C_VEL
LIN {X 0,Y 286.92,Z 920.473,A -85,B 0,C 180,E1 -17430.367,E2 -17430.367} C_VEL
LIN {X 0,Y 290.846,Z 926.914,A -85,B 0,C 180,E1 -17431.964,E2 -17431.964} C_VEL
LIN {X 0,Y 294.083,Z 932.44,A -85,B 0,C 180,E1 -17433.156,E2 -17433.156} C_VEL
LIN {X 0,Y 298.206,Z 941.27,A -85,B 0,C 180,E1 -17434.633,E2 -17434.633} C_VEL
LIN {X 0,Y 293.925,Z 985.963,A -85,B 0,C 180,E1 -17436.577,E2 -17436.577} C_VEL
LIN {X 0,Y 292.604,Z 997.089,A -85,B 0,C 180,E1 -17437.307,E2 -17437.307} C_VEL
LIN {X 0,Y 291.016,Z 1007.244,A -85,B 0,C 180,E1 -17438.205,E2 -17438.205} C_VEL
LIN {X 0,Y 289.375,Z 1016.144,A -85,B 0,C 180,E1 -17439.195,E2 -17439.195} C_VEL
LIN {X 0,Y 287.465,Z 1025.692,A -85,B 0,C 180,E1 -17440.543,E2 -17440.543} C_VEL
LIN {X 0,Y 285.341,Z 1034.19,A -85,B 0,C 180,E1 -17442.069,E2 -17442.069} C_VEL
LIN {X 0,Y 283.698,Z 1040.423,A -85,B 0,C 180,E1 -17443.449,E2 -17443.449} C_VEL
LIN {X 0,Y 281.852,Z 1046.831,A -85,B 0,C 180,E1 -17445.192,E2 -17445.192} C_VEL
LIN {X 0,Y 280.165,Z 1051.975,A -85,B 0,C 180,E1 -17446.953,E2 -17446.953} C_VEL
LIN {X 0,Y 278.634,Z 1056.692,A -85,B 0,C 180,E1 -17449.096,E2 -17449.096} C_VEL
LIN {X 0,Y 277.471,Z 1059.936,A -85,B 0,C 180,E1 -17451.259,E2 -17451.259} C_VEL
LIN {X 0,Y 276.743,Z 1061.471,A -85,B 0,C 180,E1 -17452.706,E2 -17452.706} C_VEL
LIN {X 0,Y 276.189,Z 1062.379,A -85,B 0,C 180,E1 -17454.159,E2 -17454.159} C_VEL
LIN {X 0,Y 275.848,Z 1062.735,A -85,B 0,C 180,E1 -17455.617,E2 -17455.617} C_VEL
LIN {X 0,Y 275.617,Z 1062.598,A -85,B 0,C 180,E1 -17457.077,E2 -17457.077} C_VEL
LIN {X 0,Y 275.433,Z 1061.964,A -85,B 0,C 180,E1 -17458.539,E2 -17458.539} C_VEL
LIN {X 0,Y 275.336,Z 1060.781,A -85,B 0,C 180,E1 -17460.001,E2 -17460.001} C_VEL
LIN {X 0,Y 275.375,Z 1057.846,A -85,B 0,C 180,E1 -17462.195,E2 -17462.195} C_VEL
LIN {X 0,Y 275.478,Z 1055.206,A -85,B 0,C 180,E1 -17463.658,E2 -17463.658} C_VEL
LIN {X 0,Y 275.638,Z 1049.852,A -85,B 0,C 180,E1 -17465.854,E2 -17465.854} C_VEL
LIN {X 0,Y 276.021,Z 1044.139,A -85,B 0,C 180,E1 -17467.683,E2 -17467.683} C_VEL
LIN {X 0,Y 276.473,Z 1037.019,A -85,B 0,C 180,E1 -17469.511,E2 -17469.511} C_VEL
LIN {X 0,Y 277.131,Z 1027.87,A -85,B 0,C 180,E1 -17471.335,E2 -17471.335} C_VEL
LIN {X 0,Y 277.763,Z 1019.963,A -85,B 0,C 180,E1 -17472.606,E2 -17472.606} C_VEL
LIN {X 0,Y 278.288,Z 1011.737,A -85,B 0,C 180,E1 -17473.696,E2 -17473.696} C_VEL
LIN {X 0,Y 278.981,Z 1000.626,A -85,B 0,C 180,E1 -17474.872,E2 -17474.872} C_VEL
LIN {X 0,Y 279.468,Z 990.092,A -85,B 0,C 180,E1 -17475.685,E2 -17475.685} C_VEL
LIN {X 0,Y 279.794,Z 980.531,A -85,B 0,C 180,E1 -17476.228,E2 -17476.228} C_VEL
LIN {X 0,Y 281.35,Z 927.635,A -85,B 0,C 180,E1 -17478.272,E2 -17478.272} C_VEL
LIN {X 0,Y 277.781,Z 903.176,A -85,B 0,C 180,E1 -17479.33,E2 -17479.33} C_VEL
LIN {X 0,Y 277.467,Z 900.721,A -85,B 0,C 180,E1 -17480.417,E2 -17480.417} C_VEL
LIN {X 0,Y 277.233,Z 900.763,A -85,B 0,C 180,E1 -17485.529,E2 -17485.529} C_VEL
LIN {X 0,Y 277.239,Z 900.761,A -85,B 0,C 180,E1 -17488.794,E2 -17488.794} C_VEL
LIN {X 0,Y 277.241,Z 900.76,A -85,B 0,C 180,E1 -17492.165,E2 -17492.165} C_VEL
LIN {X 0,Y 277.274,Z 900.759,A -85,B 0,C 180,E1 -17495.797,E2 -17495.797} C_VEL
LIN {X 0,Y 277.191,Z 900.766,A -85,B 0,C 180,E1 -17499.336,E2 -17499.336} C_VEL
LIN {X 0,Y 277.193,Z 900.766,A -85,B 0,C 180,E1 -17503.202,E2 -17503.202} C_VEL
LIN {X 0,Y 277.194,Z 900.765,A -85,B 0,C 180,E1 -17507.331,E2 -17507.331} C_VEL
LIN {X 0,Y 277.252,Z 900.76,A -85,B 0,C 180,E1 -17511.797,E2 -17511.797} C_VEL
LIN {X 0,Y 277.28,Z 900.76,A -85,B 0,C 180,E1 -17514.341,E2 -17514.341} C_VEL
LIN {X 0,Y 277.243,Z 900.758,A -85,B 0,C 180,E1 -17517.836,E2 -17517.836} C_VEL
LIN {X 0,Y 277.242,Z 900.761,A -85,B 0,C 180,E1 -17521.207,E2 -17521.207} C_VEL
LIN {X 0,Y 277.249,Z 900.761,A -85,B 0,C 180,E1 -17524.473,E2 -17524.473} C_VEL
LIN {X 0,Y 277.261,Z 900.757,A -85,B 0,C 180,E1 -17527.653,E2 -17527.653} C_VEL
LIN {X 0,Y 277.285,Z 900.756,A -85,B 0,C 180,E1 -17530.762,E2 -17530.762} C_VEL
LIN {X 0,Y 277.412,Z 900.742,A -85,B 0,C 180,E1 -17535.325,E2 -17535.325} C_VEL
LIN {X 0,Y 277.459,Z 900.736,A -85,B 0,C 180,E1 -17539.787,E2 -17539.787} C_VEL
LIN {X 0,Y 277.604,Z 900.714,A -85,B 0,C 180,E1 -17542.728,E2 -17542.728} C_VEL
LIN {X 0,Y 277.802,Z 900.691,A -85,B 0,C 180,E1 -17548.551,E2 -17548.551} C_VEL
LIN {X 0,Y 277.802,Z 900.691,A -85,B 0,C 180,E1 -17551.45,E2 -17551.45} C_VEL
LIN {X 0,Y 277.605,Z 900.714,A -85,B 0,C 180,E1 -17557.272,E2 -17557.272} C_VEL
LIN {X 0,Y 277.458,Z 900.736,A -85,B 0,C 180,E1 -17560.213,E2 -17560.213} C_VEL
LIN {X 0,Y 277.371,Z 900.748,A -85,B 0,C 180,E1 -17564.678,E2 -17564.678} C_VEL
LIN {X 0,Y 277.279,Z 900.757,A -85,B 0,C 180,E1 -17569.239,E2 -17569.239} C_VEL
LIN {X 0,Y 277.259,Z 900.756,A -85,B 0,C 180,E1 -17573.927,E2 -17573.927} C_VEL
LIN {X 0,Y 277.271,Z 900.759,A -85,B 0,C 180,E1 -17577.481,E2 -17577.481} C_VEL
LIN {X 0,Y 277.252,Z 900.758,A -85,B 0,C 180,E1 -17580.473,E2 -17580.473} C_VEL
LIN {X 0,Y 277.25,Z 900.76,A -85,B 0,C 180,E1 -17583.896,E2 -17583.896} C_VEL
LIN {X 0,Y 277.255,Z 900.762,A -85,B 0,C 180,E1 -17587.472,E2 -17587.472} C_VEL
LIN {X 0,Y 277.188,Z 900.766,A -85,B 0,C 180,E1 -17591.241,E2 -17591.241} C_VEL
LIN {X 0,Y 277.178,Z 900.768,A -85,B 0,C 180,E1 -17595.232,E2 -17595.232} C_VEL
LIN {X 0,Y 277.188,Z 900.767,A -85,B 0,C 180,E1 -17598.758,E2 -17598.758} C_VEL
LIN {X 0,Y 277.255,Z 900.762,A -85,B 0,C 180,E1 -17602.528,E2 -17602.528} C_VEL
LIN {X 0,Y 277.25,Z 900.761,A -85,B 0,C 180,E1 -17606.104,E2 -17606.104} C_VEL
LIN {X 0,Y 277.266,Z 900.755,A -85,B 0,C 180,E1 -17609.538,E2 -17609.538} C_VEL
LIN {X 0,Y 277.292,Z 900.759,A -85,B 0,C 180,E1 -17612.856,E2 -17612.856} C_VEL
LIN {X 0,Y 277.258,Z 900.758,A -85,B 0,C 180,E1 -17616.072,E2 -17616.072} C_VEL
LIN {X 0,Y 277.278,Z 900.756,A -85,B 0,C 180,E1 -17620.761,E2 -17620.761} C_VEL
LIN {X 0,Y 277.37,Z 900.749,A -85,B 0,C 180,E1 -17625.322,E2 -17625.322} C_VEL
LIN {X 0,Y 277.456,Z 900.736,A -85,B 0,C 180,E1 -17629.786,E2 -17629.786} C_VEL
LIN {X 0,Y 277.603,Z 900.715,A -85,B 0,C 180,E1 -17632.727,E2 -17632.727} C_VEL
LIN {X 0,Y 277.8,Z 900.69,A -85,B 0,C 180,E1 -17638.55,E2 -17638.55} C_VEL
LIN {X 0,Y 277.8,Z 900.691,A -85,B 0,C 180,E1 -17641.449,E2 -17641.449} C_VEL
LIN {X 0,Y 277.602,Z 900.713,A -85,B 0,C 180,E1 -17647.272,E2 -17647.272} C_VEL
LIN {X 0,Y 277.455,Z 900.736,A -85,B 0,C 180,E1 -17650.213,E2 -17650.213} C_VEL
LIN {X 0,Y 277.368,Z 900.748,A -85,B 0,C 180,E1 -17654.677,E2 -17654.677} C_VEL
LIN {X 0,Y 277.37,Z 900.742,A -85,B 0,C 180,E1 -17655.658,E2 -17655.658} C_VEL
LIN {X 0,Y 276.729,Z 900.827,A -85,B 0,C 180,E1 -17656.87,E2 -17656.87} C_VEL
LIN {X 0,Y 273.819,Z 901.191,A -85,B 0,C 180,E1 -17658.842,E2 -17658.842} C_VEL
LIN {X 0,Y 271.321,Z 901.499,A -85,B 0,C 180,E1 -17660.445,E2 -17660.445} C_VEL
LIN {X 0,Y 270.246,Z 901.632,A -85,B 0,C 180,E1 -17661.689,E2 -17661.689} C_VEL
LIN {X 0,Y 270.159,Z 901.642,A -85,B 0,C 180,E1 -17662.111,E2 -17662.111} C_VEL
LIN {X 0,Y 270.194,Z 901.636,A -85,B 0,C 180,E1 -17666.243,E2 -17666.243} C_VEL
LIN {X 0,Y 270.183,Z 901.642,A -85,B 0,C 180,E1 -17669.618,E2 -17669.618} C_VEL
LIN {X 0,Y 270.215,Z 901.637,A -85,B 0,C 180,E1 -17673.665,E2 -17673.665} C_VEL
LIN {X 0,Y 270.207,Z 901.636,A -85,B 0,C 180,E1 -17676.742,E2 -17676.742} C_VEL
LIN {X 0,Y 270.147,Z 901.644,A -85,B 0,C 180,E1 -17680.57,E2 -17680.57} C_VEL
LIN {X 0,Y 270.128,Z 901.645,A -85,B 0,C 180,E1 -17684.625,E2 -17684.625} C_VEL
LIN {X 0,Y 270.15,Z 901.644,A -85,B 0,C 180,E1 -17687.437,E2 -17687.437} C_VEL
LIN {X 0,Y 270.191,Z 901.637,A -85,B 0,C 180,E1 -17691.371,E2 -17691.371} C_VEL
LIN {X 0,Y 270.196,Z 901.638,A -85,B 0,C 180,E1 -17695.093,E2 -17695.093} C_VEL
LIN {X 0,Y 270.183,Z 901.64,A -85,B 0,C 180,E1 -17699.136,E2 -17699.136} C_VEL
LIN {X 0,Y 270.347,Z 901.794,A -85,B 0,C 180,E1 -17701.815,E2 -17701.815} C_VEL
LIN {X 0,Y 272.218,Z 911.816,A -85,B 0,C 180,E1 -17705.601,E2 -17705.601} C_VEL
LIN {X 0,Y 272.142,Z 915.146,A -85,B 0,C 180,E1 -17706.807,E2 -17706.807} C_VEL
LIN {X 0,Y 270.856,Z 925.192,A -85,B 0,C 180,E1 -17710.385,E2 -17710.385} C_VEL
LIN {X 0,Y 272.079,Z 943.917,A -85,B 0,C 180,E1 -17711.187,E2 -17711.187} C_VEL
LIN {X 0,Y 273.963,Z 962.297,A -85,B 0,C 180,E1 -17711.974,E2 -17711.974} C_VEL
LIN {X 0,Y 272.772,Z 1004.001,A -85,B 0,C 180,E1 -17713.68,E2 -17713.68} C_VEL
LIN {X 0,Y 272.043,Z 1016.157,A -85,B 0,C 180,E1 -17714.453,E2 -17714.453} C_VEL
LIN {X 0,Y 271.553,Z 1026.406,A -85,B 0,C 180,E1 -17715.384,E2 -17715.384} C_VEL
LIN {X 0,Y 270.877,Z 1035.95,A -85,B 0,C 180,E1 -17716.496,E2 -17716.496} C_VEL
LIN {X 0,Y 270.135,Z 1046.034,A -85,B 0,C 180,E1 -17717.987,E2 -17717.987} C_VEL
LIN {X 0,Y 269.584,Z 1053.975,A -85,B 0,C 180,E1 -17719.485,E2 -17719.485} C_VEL
LIN {X 0,Y 269.156,Z 1060.538,A -85,B 0,C 180,E1 -17720.986,E2 -17720.986} C_VEL
LIN {X 0,Y 268.897,Z 1066.001,A -85,B 0,C 180,E1 -17722.491,E2 -17722.491} C_VEL
LIN {X 0,Y 268.672,Z 1070.521,A -85,B 0,C 180,E1 -17723.994,E2 -17723.994} C_VEL
LIN {X 0,Y 268.56,Z 1074.249,A -85,B 0,C 180,E1 -17725.497,E2 -17725.497} C_VEL
LIN {X 0,Y 268.379,Z 1077.256,A -85,B 0,C 180,E1 -17726.998,E2 -17726.998} C_VEL
LIN {X 0,Y 268.341,Z 1079.595,A -85,B 0,C 180,E1 -17728.499,E2 -17728.499} C_VEL
LIN {X 0,Y 268.362,Z 1081.267,A -85,B 0,C 180,E1 -17730,E2 -17730} C_VEL
LIN {X 0,Y 268.236,Z 1082.348,A -85,B 0,C 180,E1 -17731.501,E2 -17731.501} C_VEL
LIN {X 0,Y 268.29,Z 1082.916,A -85,B 0,C 180,E1 -17733.003,E2 -17733.003} C_VEL
LIN {X 0,Y 268.257,Z 1082.981,A -85,B 0,C 180,E1 -17734.508,E2 -17734.508} C_VEL
LIN {X 0,Y 268.389,Z 1082.484,A -85,B 0,C 180,E1 -17736.012,E2 -17736.012} C_VEL
LIN {X 0,Y 268.664,Z 1081.389,A -85,B 0,C 180,E1 -17737.515,E2 -17737.515} C_VEL
LIN {X 0,Y 269.424,Z 1078.858,A -85,B 0,C 180,E1 -17739.762,E2 -17739.762} C_VEL
LIN {X 0,Y 270.644,Z 1075.019,A -85,B 0,C 180,E1 -17741.99,E2 -17741.99} C_VEL
LIN {X 0,Y 272.265,Z 1069.713,A -85,B 0,C 180,E1 -17744.195,E2 -17744.195} C_VEL
LIN {X 0,Y 273.848,Z 1064.09,A -85,B 0,C 180,E1 -17746.015,E2 -17746.015} C_VEL
LIN {X 0,Y 275.906,Z 1057.235,A -85,B 0,C 180,E1 -17747.798,E2 -17747.798} C_VEL
LIN {X 0,Y 278.302,Z 1048.695,A -85,B 0,C 180,E1 -17749.548,E2 -17749.548} C_VEL
LIN {X 0,Y 280.434,Z 1040.186,A -85,B 0,C 180,E1 -17750.923,E2 -17750.923} C_VEL
LIN {X 0,Y 282.187,Z 1032.58,A -85,B 0,C 180,E1 -17751.936,E2 -17751.936} C_VEL
LIN {X 0,Y 284.242,Z 1023.423,A -85,B 0,C 180,E1 -17752.919,E2 -17752.919} C_VEL
LIN {X 0,Y 286.435,Z 1011.895,A -85,B 0,C 180,E1 -17753.881,E2 -17753.881} C_VEL
LIN {X 0,Y 288.15,Z 999.383,A -85,B 0,C 180,E1 -17754.614,E2 -17754.614} C_VEL
LIN {X 0,Y 291.256,Z 967.036,A -85,B 0,C 180,E1 -17756.073,E2 -17756.073} C_VEL
LIN {X 0,Y 290.567,Z 958.252,A -85,B 0,C 180,E1 -17756.802,E2 -17756.802} C_VEL
LIN {X 0,Y 288.598,Z 945.731,A -85,B 0,C 180,E1 -17758.137,E2 -17758.137} C_VEL
LIN {X 0,Y 287.125,Z 941.063,A -85,B 0,C 180,E1 -17758.86,E2 -17758.86} C_VEL
LIN {X 0,Y 284.565,Z 935.75,A -85,B 0,C 180,E1 -17759.984,E2 -17759.984} C_VEL
LIN {X 0,Y 281.864,Z 930.502,A -85,B 0,C 180,E1 -17761.251,E2 -17761.251} C_VEL
LIN {X 0,Y 279.305,Z 925.523,A -85,B 0,C 180,E1 -17762.632,E2 -17762.632} C_VEL
LIN {X 0,Y 275.697,Z 920.065,A -85,B 0,C 180,E1 -17764.721,E2 -17764.721} C_VEL
LIN {X 0,Y 274.934,Z 918.234,A -85,B 0,C 180,E1 -17765.392,E2 -17765.392} C_VEL
LIN {X 0,Y 274.215,Z 915.685,A -85,B 0,C 180,E1 -17767.96,E2 -17767.96} C_VEL
LIN {X 0,Y 273.808,Z 914.078,A -85,B 0,C 180,E1 -17769.918,E2 -17769.918} C_VEL
LIN {X 0,Y 273.437,Z 912.795,A -85,B 0,C 180,E1 -17771.933,E2 -17771.933} C_VEL
LIN {X 0,Y 272.995,Z 911.258,A -85,B 0,C 180,E1 -17775.966,E2 -17775.966} C_VEL
LIN {X 0,Y 272.946,Z 910.993,A -85,B 0,C 180,E1 -17778.306,E2 -17778.306} C_VEL
LIN {X 0,Y 273.021,Z 911.475,A -85,B 0,C 180,E1 -17781.845,E2 -17781.845} C_VEL
LIN {X 0,Y 273.285,Z 912.329,A -85,B 0,C 180,E1 -17783.912,E2 -17783.912} C_VEL
LIN {X 0,Y 275.792,Z 915.869,A -85,B 0,C 180,E1 -17785.761,E2 -17785.761} C_VEL
LIN {X 0,Y 277.645,Z 917.818,A -85,B 0,C 180,E1 -17786.835,E2 -17786.835} C_VEL
LIN {X 0,Y 280.007,Z 921.313,A -85,B 0,C 180,E1 -17788.155,E2 -17788.155} C_VEL
LIN {X 0,Y 281.268,Z 922.874,A -85,B 0,C 180,E1 -17788.771,E2 -17788.771} C_VEL
LIN {X 0,Y 284.26,Z 927.485,A -85,B 0,C 180,E1 -17790.173,E2 -17790.173} C_VEL
LIN {X 0,Y 287.005,Z 932.031,A -85,B 0,C 180,E1 -17791.361,E2 -17791.361} C_VEL
LIN {X 0,Y 290.556,Z 938.546,A -85,B 0,C 180,E1 -17792.767,E2 -17792.767} C_VEL
LIN {X 0,Y 293.126,Z 944.094,A -85,B 0,C 180,E1 -17793.737,E2 -17793.737} C_VEL
LIN {X 0,Y 288.515,Z 987.973,A -85,B 0,C 180,E1 -17795.729,E2 -17795.729} C_VEL
LIN {X 0,Y 286.951,Z 999.477,A -85,B 0,C 180,E1 -17796.548,E2 -17796.548} C_VEL
LIN {X 0,Y 285.076,Z 1010.003,A -85,B 0,C 180,E1 -17797.535,E2 -17797.535} C_VEL
LIN {X 0,Y 282.849,Z 1020.8,A -85,B 0,C 180,E1 -17798.883,E2 -17798.883} C_VEL
LIN {X 0,Y 280.79,Z 1029.354,A -85,B 0,C 180,E1 -17800.252,E2 -17800.252} C_VEL
LIN {X 0,Y 278.87,Z 1036.472,A -85,B 0,C 180,E1 -17801.639,E2 -17801.639} C_VEL
LIN {X 0,Y 276.734,Z 1043.752,A -85,B 0,C 180,E1 -17803.399,E2 -17803.399} C_VEL
LIN {X 0,Y 274.798,Z 1049.564,A -85,B 0,C 180,E1 -17805.183,E2 -17805.183} C_VEL
LIN {X 0,Y 273.399,Z 1053.367,A -85,B 0,C 180,E1 -17806.624,E2 -17806.624} C_VEL
LIN {X 0,Y 271.746,Z 1057.731,A -85,B 0,C 180,E1 -17808.816,E2 -17808.816} C_VEL
LIN {X 0,Y 270.941,Z 1059.922,A -85,B 0,C 180,E1 -17810.295,E2 -17810.295} C_VEL
LIN {X 0,Y 269.753,Z 1062.078,A -85,B 0,C 180,E1 -17812.516,E2 -17812.516} C_VEL
LIN {X 0,Y 269.168,Z 1062.922,A -85,B 0,C 180,E1 -17814.006,E2 -17814.006} C_VEL
LIN {X 0,Y 268.798,Z 1063.146,A -85,B 0,C 180,E1 -17815.502,E2 -17815.502} C_VEL
LIN {X 0,Y 268.549,Z 1062.833,A -85,B 0,C 180,E1 -17817,E2 -17817} C_VEL
LIN {X 0,Y 268.357,Z 1062.022,A -85,B 0,C 180,E1 -17818.5,E2 -17818.5} C_VEL
LIN {X 0,Y 268.257,Z 1060.701,A -85,B 0,C 180,E1 -17820.001,E2 -17820.001} C_VEL
LIN {X 0,Y 268.263,Z 1058.828,A -85,B 0,C 180,E1 -17821.502,E2 -17821.502} C_VEL
LIN {X 0,Y 268.398,Z 1054.759,A -85,B 0,C 180,E1 -17823.754,E2 -17823.754} C_VEL
LIN {X 0,Y 268.471,Z 1050.969,A -85,B 0,C 180,E1 -17825.363,E2 -17825.363} C_VEL
LIN {X 0,Y 268.799,Z 1045.887,A -85,B 0,C 180,E1 -17827.097,E2 -17827.097} C_VEL
LIN {X 0,Y 269.159,Z 1040.393,A -85,B 0,C 180,E1 -17828.636,E2 -17828.636} C_VEL
LIN {X 0,Y 269.576,Z 1033.936,A -85,B 0,C 180,E1 -17830.136,E2 -17830.136} C_VEL
LIN {X 0,Y 270.181,Z 1026.163,A -85,B 0,C 180,E1 -17831.631,E2 -17831.631} C_VEL
LIN {X 0,Y 270.858,Z 1016.636,A -85,B 0,C 180,E1 -17833.123,E2 -17833.123} C_VEL
LIN {X 0,Y 271.597,Z 1005.798,A -85,B 0,C 180,E1 -17834.423,E2 -17834.423} C_VEL
LIN {X 0,Y 272.161,Z 995.889,A -85,B 0,C 180,E1 -17835.349,E2 -17835.349} C_VEL
LIN {X 0,Y 272.439,Z 986.772,A -85,B 0,C 180,E1 -17836.005,E2 -17836.005} C_VEL
LIN {X 0,Y 273.042,Z 972.727,A -85,B 0,C 180,E1 -17836.689,E2 -17836.689} C_VEL
LIN {X 0,Y 274.3,Z 928.42,A -85,B 0,C 180,E1 -17838.429,E2 -17838.429} C_VEL
LIN {X 0,Y 270.673,Z 903.331,A -85,B 0,C 180,E1 -17839.595,E2 -17839.595} C_VEL
LIN {X 0,Y 270.45,Z 901.596,A -85,B 0,C 180,E1 -17840.375,E2 -17840.375} C_VEL
LIN {X 0,Y 270.178,Z 901.641,A -85,B 0,C 180,E1 -17844.596,E2 -17844.596} C_VEL
LIN {X 0,Y 270.197,Z 901.637,A -85,B 0,C 180,E1 -17847.918,E2 -17847.918} C_VEL
LIN {X 0,Y 270.175,Z 901.643,A -85,B 0,C 180,E1 -17851.35,E2 -17851.35} C_VEL
LIN {X 0,Y 270.199,Z 901.638,A -85,B 0,C 180,E1 -17854.907,E2 -17854.907} C_VEL
LIN {X 0,Y 270.169,Z 901.639,A -85,B 0,C 180,E1 -17858.703,E2 -17858.703} C_VEL
LIN {X 0,Y 270.15,Z 901.644,A -85,B 0,C 180,E1 -17863.246,E2 -17863.246} C_VEL
LIN {X 0,Y 270.153,Z 901.642,A -85,B 0,C 180,E1 -17867.438,E2 -17867.438} C_VEL
LIN {X 0,Y 270.195,Z 901.637,A -85,B 0,C 180,E1 -17871.372,E2 -17871.372} C_VEL
LIN {X 0,Y 270.2,Z 901.637,A -85,B 0,C 180,E1 -17875.095,E2 -17875.095} C_VEL
LIN {X 0,Y 270.187,Z 901.639,A -85,B 0,C 180,E1 -17879.137,E2 -17879.137} C_VEL
LIN {X 0,Y 270.226,Z 901.635,A -85,B 0,C 180,E1 -17882.164,E2 -17882.164} C_VEL
LIN {X 0,Y 270.231,Z 901.633,A -85,B 0,C 180,E1 -17885.543,E2 -17885.543} C_VEL
LIN {X 0,Y 270.226,Z 901.634,A -85,B 0,C 180,E1 -17890.239,E2 -17890.239} C_VEL
LIN {X 0,Y 270.372,Z 901.617,A -85,B 0,C 180,E1 -17894.934,E2 -17894.934} C_VEL
LIN {X 0,Y 270.41,Z 901.616,A -85,B 0,C 180,E1 -17899.518,E2 -17899.518} C_VEL
LIN {X 0,Y 270.566,Z 901.591,A -85,B 0,C 180,E1 -17902.538,E2 -17902.538} C_VEL
LIN {X 0,Y 270.766,Z 901.567,A -85,B 0,C 180,E1 -17908.513,E2 -17908.513} C_VEL
LIN {X 0,Y 270.766,Z 901.568,A -85,B 0,C 180,E1 -17911.488,E2 -17911.488} C_VEL
LIN {X 0,Y 270.566,Z 901.591,A -85,B 0,C 180,E1 -17917.463,E2 -17917.463} C_VEL
LIN {X 0,Y 270.409,Z 901.616,A -85,B 0,C 180,E1 -17920.483,E2 -17920.483} C_VEL
LIN {X 0,Y 270.342,Z 901.621,A -85,B 0,C 180,E1 -17925.068,E2 -17925.068} C_VEL
LIN {X 0,Y 270.223,Z 901.634,A -85,B 0,C 180,E1 -17929.762,E2 -17929.762} C_VEL
LIN {X 0,Y 270.186,Z 901.638,A -85,B 0,C 180,E1 -17934.436,E2 -17934.436} C_VEL
LIN {X 0,Y 270.2,Z 901.638,A -85,B 0,C 180,E1 -17937.917,E2 -17937.917} C_VEL
LIN {X 0,Y 270.178,Z 901.643,A -85,B 0,C 180,E1 -17941.349,E2 -17941.349} C_VEL
LIN {X 0,Y 270.202,Z 901.637,A -85,B 0,C 180,E1 -17944.906,E2 -17944.906} C_VEL
LIN {X 0,Y 270.202,Z 901.636,A -85,B 0,C 180,E1 -17948.71,E2 -17948.71} C_VEL
LIN {X 0,Y 270.152,Z 901.642,A -85,B 0,C 180,E1 -17953.245,E2 -17953.245} C_VEL
LIN {X 0,Y 270.155,Z 901.643,A -85,B 0,C 180,E1 -17957.437,E2 -17957.437} C_VEL
LIN {X 0,Y 270.196,Z 901.636,A -85,B 0,C 180,E1 -17961.371,E2 -17961.371} C_VEL
LIN {X 0,Y 270.201,Z 901.638,A -85,B 0,C 180,E1 -17965.093,E2 -17965.093} C_VEL
LIN {X 0,Y 270.188,Z 901.638,A -85,B 0,C 180,E1 -17969.136,E2 -17969.136} C_VEL
LIN {X 0,Y 270.203,Z 901.637,A -85,B 0,C 180,E1 -17972.172,E2 -17972.172} C_VEL
LIN {X 0,Y 270.185,Z 901.639,A -85,B 0,C 180,E1 -17975.564,E2 -17975.564} C_VEL
LIN {X 0,Y 270.222,Z 901.633,A -85,B 0,C 180,E1 -17980.238,E2 -17980.238} C_VEL
LIN {X 0,Y 270.34,Z 901.622,A -85,B 0,C 180,E1 -17984.931,E2 -17984.931} C_VEL
LIN {X 0,Y 270.389,Z 901.617,A -85,B 0,C 180,E1 -17989.516,E2 -17989.516} C_VEL
LIN {X 0,Y 270.565,Z 901.592,A -85,B 0,C 180,E1 -17992.537,E2 -17992.537} C_VEL
LIN {X 0,Y 270.764,Z 901.567,A -85,B 0,C 180,E1 -17998.512,E2 -17998.512} C_VEL
LIN {X 0,Y 270.763,Z 901.568,A -85,B 0,C 180,E1 -18001.487,E2 -18001.487} C_VEL
LIN {X 0,Y 270.564,Z 901.59,A -85,B 0,C 180,E1 -18007.462,E2 -18007.462} C_VEL
LIN {X 0,Y 270.406,Z 901.617,A -85,B 0,C 180,E1 -18010.482,E2 -18010.482} C_VEL
LIN {X 0,Y 270.338,Z 901.62,A -85,B 0,C 180,E1 -18015.068,E2 -18015.068} C_VEL
LIN {X 0,Y 270.22,Z 901.635,A -85,B 0,C 180,E1 -18019.761,E2 -18019.761} C_VEL
LIN {X 0,Y 270.159,Z 901.642,A -85,B 0,C 180,E1 -18022.111,E2 -18022.111} C_VEL
LIN {X 0,Y 269.508,Z 901.728,A -85,B 0,C 180,E1 -18023.354,E2 -18023.354} C_VEL
LIN {X 0,Y 266.714,Z 902.082,A -85,B 0,C 180,E1 -18025.382,E2 -18025.382} C_VEL
LIN {X 0,Y 264.312,Z 902.381,A -85,B 0,C 180,E1 -18027.03,E2 -18027.03} C_VEL
LIN {X 0,Y 263.241,Z 902.508,A -85,B 0,C 180,E1 -18028.305,E2 -18028.305} C_VEL
LIN {X 0,Y 263.132,Z 902.518,A -85,B 0,C 180,E1 -18028.738,E2 -18028.738} C_VEL
LIN {X 0,Y 263.128,Z 902.517,A -85,B 0,C 180,E1 -18032.288,E2 -18032.288} C_VEL
LIN {X 0,Y 263.174,Z 902.512,A -85,B 0,C 180,E1 -18036.76,E2 -18036.76} C_VEL
LIN {X 0,Y 263.091,Z 902.527,A -85,B 0,C 180,E1 -18039.874,E2 -18039.874} C_VEL
LIN {X 0,Y 263.076,Z 902.527,A -85,B 0,C 180,E1 -18043.993,E2 -18043.993} C_VEL
LIN {X 0,Y 263.108,Z 902.524,A -85,B 0,C 180,E1 -18048.41,E2 -18048.41} C_VEL
LIN {X 0,Y 263.146,Z 902.518,A -85,B 0,C 180,E1 -18052.1,E2 -18052.1} C_VEL
LIN {X 0,Y 263.15,Z 902.516,A -85,B 0,C 180,E1 -18055.885,E2 -18055.885} C_VEL
LIN {X 0,Y 263.143,Z 902.516,A -85,B 0,C 180,E1 -18059.505,E2 -18059.505} C_VEL
LIN {X 0,Y 263.312,Z 902.559,A -85,B 0,C 180,E1 -18061.737,E2 -18061.737} C_VEL
LIN {X 0,Y 265.191,Z 912.9,A -85,B 0,C 180,E1 -18065.746,E2 -18065.746} C_VEL
LIN {X 0,Y 264.682,Z 918.358,A -85,B 0,C 180,E1 -18067.767,E2 -18067.767} C_VEL
LIN {X 0,Y 263.834,Z 924.83,A -85,B 0,C 180,E1 -18070.145,E2 -18070.145} C_VEL
LIN {X 0,Y 264.827,Z 941.568,A -85,B 0,C 180,E1 -18070.903,E2 -18070.903} C_VEL
LIN {X 0,Y 266.862,Z 963.226,A -85,B 0,C 180,E1 -18071.863,E2 -18071.863} C_VEL
LIN {X 0,Y 265.68,Z 1004.254,A -85,B 0,C 180,E1 -18073.627,E2 -18073.627} C_VEL
LIN {X 0,Y 264.906,Z 1017.153,A -85,B 0,C 180,E1 -18074.516,E2 -18074.516} C_VEL
LIN {X 0,Y 264.457,Z 1026.194,A -85,B 0,C 180,E1 -18075.376,E2 -18075.376} C_VEL
LIN {X 0,Y 263.799,Z 1035.691,A -85,B 0,C 180,E1 -18076.519,E2 -18076.519} C_VEL
LIN {X 0,Y 263.041,Z 1045.759,A -85,B 0,C 180,E1 -18078.049,E2 -18078.049} C_VEL
LIN {X 0,Y 262.508,Z 1053.701,A -85,B 0,C 180,E1 -18079.588,E2 -18079.588} C_VEL
LIN {X 0,Y 262.085,Z 1060.261,A -85,B 0,C 180,E1 -18081.13,E2 -18081.13} C_VEL
LIN {X 0,Y 261.822,Z 1065.844,A -85,B 0,C 180,E1 -18082.713,E2 -18082.713} C_VEL
LIN {X 0,Y 261.604,Z 1070.499,A -85,B 0,C 180,E1 -18084.319,E2 -18084.319} C_VEL
LIN {X 0,Y 261.457,Z 1074.742,A -85,B 0,C 180,E1 -18086.146,E2 -18086.146} C_VEL
LIN {X 0,Y 261.323,Z 1077.529,A -85,B 0,C 180,E1 -18087.688,E2 -18087.688} C_VEL
LIN {X 0,Y 261.313,Z 1080.509,A -85,B 0,C 180,E1 -18090,E2 -18090} C_VEL
LIN {X 0,Y 261.164,Z 1081.758,A -85,B 0,C 180,E1 -18091.542,E2 -18091.542} C_VEL
LIN {X 0,Y 261.221,Z 1082.505,A -85,B 0,C 180,E1 -18093.084,E2 -18093.084} C_VEL
LIN {X 0,Y 261.226,Z 1082.478,A -85,B 0,C 180,E1 -18095.476,E2 -18095.476} C_VEL
LIN {X 0,Y 261.607,Z 1081.336,A -85,B 0,C 180,E1 -18097.719,E2 -18097.719} C_VEL
LIN {X 0,Y 262.124,Z 1079.935,A -85,B 0,C 180,E1 -18099.257,E2 -18099.257} C_VEL
LIN {X 0,Y 263.229,Z 1076.751,A -85,B 0,C 180,E1 -18101.551,E2 -18101.551} C_VEL
LIN {X 0,Y 264.824,Z 1072.272,A -85,B 0,C 180,E1 -18103.818,E2 -18103.818} C_VEL
LIN {X 0,Y 266.799,Z 1066.394,A -85,B 0,C 180,E1 -18106.057,E2 -18106.057} C_VEL
LIN {X 0,Y 268.804,Z 1060.07,A -85,B 0,C 180,E1 -18107.891,E2 -18107.891} C_VEL
LIN {X 0,Y 270.692,Z 1053.967,A -85,B 0,C 180,E1 -18109.331,E2 -18109.331} C_VEL
LIN {X 0,Y 272.833,Z 1046.762,A -85,B 0,C 180,E1 -18110.744,E2 -18110.744} C_VEL
LIN {X 0,Y 275.174,Z 1038.101,A -85,B 0,C 180,E1 -18112.13,E2 -18112.13} C_VEL
LIN {X 0,Y 277.931,Z 1027.334,A -85,B 0,C 180,E1 -18113.47,E2 -18113.47} C_VEL
LIN {X 0,Y 280.18,Z 1016.781,A -85,B 0,C 180,E1 -18114.449,E2 -18114.449} C_VEL
LIN {X 0,Y 282.018,Z 1006.4,A -85,B 0,C 180,E1 -18115.209,E2 -18115.209} C_VEL
LIN {X 0,Y 283.847,Z 992.591,A -85,B 0,C 180,E1 -18115.929,E2 -18115.929} C_VEL
LIN {X 0,Y 286.285,Z 968.25,A -85,B 0,C 180,E1 -18117.054,E2 -18117.054} C_VEL
LIN {X 0,Y 285.643,Z 959.783,A -85,B 0,C 180,E1 -18117.815,E2 -18117.815} C_VEL
LIN {X 0,Y 284.013,Z 948.569,A -85,B 0,C 180,E1 -18119.082,E2 -18119.082} C_VEL
LIN {X 0,Y 282.283,Z 944.127,A -85,B 0,C 180,E1 -18119.935,E2 -18119.935} C_VEL
LIN {X 0,Y 280.635,Z 940.464,A -85,B 0,C 180,E1 -18120.748,E2 -18120.748} C_VEL
LIN {X 0,Y 278.557,Z 936.11,A -85,B 0,C 180,E1 -18121.841,E2 -18121.841} C_VEL
LIN {X 0,Y 275.776,Z 930.767,A -85,B 0,C 180,E1 -18123.424,E2 -18123.424} C_VEL
LIN {X 0,Y 272.835,Z 925.842,A -85,B 0,C 180,E1 -18125.335,E2 -18125.335} C_VEL
LIN {X 0,Y 272.17,Z 924.421,A -85,B 0,C 180,E1 -18125.89,E2 -18125.89} C_VEL
LIN {X 0,Y 268.246,Z 918.746,A -85,B 0,C 180,E1 -18129.494,E2 -18129.494} C_VEL
LIN {X 0,Y 267.193,Z 916.343,A -85,B 0,C 180,E1 -18131.352,E2 -18131.352} C_VEL
LIN {X 0,Y 266.708,Z 914.669,A -85,B 0,C 180,E1 -18135.355,E2 -18135.355} C_VEL
LIN {X 0,Y 266.648,Z 914.265,A -85,B 0,C 180,E1 -18138.006,E2 -18138.006} C_VEL
LIN {X 0,Y 268.833,Z 917.18,A -85,B 0,C 180,E1 -18141.654,E2 -18141.654} C_VEL
LIN {X 0,Y 271.016,Z 918.986,A -85,B 0,C 180,E1 -18143.608,E2 -18143.608} C_VEL
LIN {X 0,Y 273.839,Z 922.835,A -85,B 0,C 180,E1 -18145.736,E2 -18145.736} C_VEL
LIN {X 0,Y 274.916,Z 924.068,A -85,B 0,C 180,E1 -18146.381,E2 -18146.381} C_VEL
LIN {X 0,Y 277.511,Z 927.849,A -85,B 0,C 180,E1 -18147.908,E2 -18147.908} C_VEL
LIN {X 0,Y 281.047,Z 933.398,A -85,B 0,C 180,E1 -18149.71,E2 -18149.71} C_VEL
LIN {X 0,Y 284.771,Z 939.894,A -85,B 0,C 180,E1 -18151.39,E2 -18151.39} C_VEL
LIN {X 0,Y 288.108,Z 946.936,A -85,B 0,C 180,E1 -18152.789,E2 -18152.789} C_VEL
LIN {X 0,Y 283.518,Z 987.81,A -85,B 0,C 180,E1 -18154.698,E2 -18154.698} C_VEL
LIN {X 0,Y 282.196,Z 997.265,A -85,B 0,C 180,E1 -18155.346,E2 -18155.346} C_VEL
LIN {X 0,Y 280.239,Z 1008.052,A -85,B 0,C 180,E1 -18156.344,E2 -18156.344} C_VEL
LIN {X 0,Y 278.302,Z 1016.839,A -85,B 0,C 180,E1 -18157.35,E2 -18157.35} C_VEL
LIN {X 0,Y 276.042,Z 1026.327,A -85,B 0,C 180,E1 -18158.728,E2 -18158.728} C_VEL
LIN {X 0,Y 273.397,Z 1035.589,A -85,B 0,C 180,E1 -18160.478,E2 -18160.478} C_VEL
LIN {X 0,Y 271.008,Z 1043.026,A -85,B 0,C 180,E1 -18162.26,E2 -18162.26} C_VEL
LIN {X 0,Y 268.505,Z 1050.157,A -85,B 0,C 180,E1 -18164.438,E2 -18164.438} C_VEL
LIN {X 0,Y 266.641,Z 1054.69,A -85,B 0,C 180,E1 -18166.278,E2 -18166.278} C_VEL
LIN {X 0,Y 265.414,Z 1057.602,A -85,B 0,C 180,E1 -18167.771,E2 -18167.771} C_VEL
LIN {X 0,Y 264.017,Z 1060.752,A -85,B 0,C 180,E1 -18170.038,E2 -18170.038} C_VEL
LIN {X 0,Y 262.767,Z 1062.7,A -85,B 0,C 180,E1 -18172.315,E2 -18172.315} C_VEL
LIN {X 0,Y 262.128,Z 1063.369,A -85,B 0,C 180,E1 -18173.844,E2 -18173.844} C_VEL
LIN {X 0,Y 261.751,Z 1063.52,A -85,B 0,C 180,E1 -18175.381,E2 -18175.381} C_VEL
LIN {X 0,Y 261.483,Z 1063.061,A -85,B 0,C 180,E1 -18176.919,E2 -18176.919} C_VEL
LIN {X 0,Y 261.283,Z 1062.071,A -85,B 0,C 180,E1 -18178.459,E2 -18178.459} C_VEL
LIN {X 0,Y 261.163,Z 1059.642,A -85,B 0,C 180,E1 -18180.772,E2 -18180.772} C_VEL
LIN {X 0,Y 261.277,Z 1055.887,A -85,B 0,C 180,E1 -18183.085,E2 -18183.085} C_VEL
LIN {X 0,Y 261.369,Z 1050.934,A -85,B 0,C 180,E1 -18185.255,E2 -18185.255} C_VEL
LIN {X 0,Y 261.69,Z 1046.107,A -85,B 0,C 180,E1 -18186.942,E2 -18186.942} C_VEL
LIN {X 0,Y 262.029,Z 1040.757,A -85,B 0,C 180,E1 -18188.484,E2 -18188.484} C_VEL
LIN {X 0,Y 262.462,Z 1034.302,A -85,B 0,C 180,E1 -18190.024,E2 -18190.024} C_VEL
LIN {X 0,Y 263.046,Z 1026.522,A -85,B 0,C 180,E1 -18191.56,E2 -18191.56} C_VEL
LIN {X 0,Y 263.77,Z 1017.017,A -85,B 0,C 180,E1 -18193.091,E2 -18193.091} C_VEL
LIN {X 0,Y 264.476,Z 1006.187,A -85,B 0,C 180,E1 -18194.427,E2 -18194.427} C_VEL
LIN {X 0,Y 265.034,Z 996.301,A -85,B 0,C 180,E1 -18195.378,E2 -18195.378} C_VEL
LIN {X 0,Y 265.312,Z 988.681,A -85,B 0,C 180,E1 -18195.953,E2 -18195.953} C_VEL
LIN {X 0,Y 265.776,Z 977.782,A -85,B 0,C 180,E1 -18196.565,E2 -18196.565} C_VEL
LIN {X 0,Y 267.243,Z 928.926,A -85,B 0,C 180,E1 -18198.595,E2 -18198.595} C_VEL
LIN {X 0,Y 263.558,Z 903.69,A -85,B 0,C 180,E1 -18199.782,E2 -18199.782} C_VEL
LIN {X 0,Y 263.392,Z 902.475,A -85,B 0,C 180,E1 -18200.404,E2 -18200.404} C_VEL
LIN {X 0,Y 263.127,Z 902.522,A -85,B 0,C 180,E1 -18205.301,E2 -18205.301} C_VEL
LIN {X 0,Y 263.134,Z 902.518,A -85,B 0,C 180,E1 -18208.736,E2 -18208.736} C_VEL
LIN {X 0,Y 263.13,Z 902.517,A -85,B 0,C 180,E1 -18212.29,E2 -18212.29} C_VEL
LIN {X 0,Y 263.156,Z 902.516,A -85,B 0,C 180,E1 -18215.984,E2 -18215.984} C_VEL
LIN {X 0,Y 263.074,Z 902.528,A -85,B 0,C 180,E1 -18219.879,E2 -18219.879} C_VEL
LIN {X 0,Y 263.078,Z 902.529,A -85,B 0,C 180,E1 -18223.995,E2 -18223.995} C_VEL
LIN {X 0,Y 263.111,Z 902.521,A -85,B 0,C 180,E1 -18228.411,E2 -18228.411} C_VEL
LIN {X 0,Y 263.15,Z 902.518,A -85,B 0,C 180,E1 -18232.102,E2 -18232.102} C_VEL
LIN {X 0,Y 263.154,Z 902.515,A -85,B 0,C 180,E1 -18235.886,E2 -18235.886} C_VEL
LIN {X 0,Y 263.129,Z 902.517,A -85,B 0,C 180,E1 -18239.504,E2 -18239.504} C_VEL
LIN {X 0,Y 263.145,Z 902.519,A -85,B 0,C 180,E1 -18242.998,E2 -18242.998} C_VEL
LIN {X 0,Y 263.147,Z 902.515,A -85,B 0,C 180,E1 -18246.384,E2 -18246.384} C_VEL
LIN {X 0,Y 263.212,Z 902.508,A -85,B 0,C 180,E1 -18249.689,E2 -18249.689} C_VEL
LIN {X 0,Y 263.314,Z 902.494,A -85,B 0,C 180,E1 -18254.52,E2 -18254.52} C_VEL
LIN {X 0,Y 263.35,Z 902.493,A -85,B 0,C 180,E1 -18259.234,E2 -18259.234} C_VEL
LIN {X 0,Y 263.53,Z 902.468,A -85,B 0,C 180,E1 -18262.337,E2 -18262.337} C_VEL
LIN {X 0,Y 263.728,Z 902.444,A -85,B 0,C 180,E1 -18268.473,E2 -18268.473} C_VEL
LIN {X 0,Y 263.728,Z 902.444,A -85,B 0,C 180,E1 -18271.527,E2 -18271.527} C_VEL
LIN {X 0,Y 263.531,Z 902.468,A -85,B 0,C 180,E1 -18277.663,E2 -18277.663} C_VEL
LIN {X 0,Y 263.348,Z 902.493,A -85,B 0,C 180,E1 -18280.767,E2 -18280.767} C_VEL
LIN {X 0,Y 263.293,Z 902.497,A -85,B 0,C 180,E1 -18285.482,E2 -18285.482} C_VEL
LIN {X 0,Y 263.211,Z 902.508,A -85,B 0,C 180,E1 -18290.311,E2 -18290.311} C_VEL
LIN {X 0,Y 263.13,Z 902.521,A -85,B 0,C 180,E1 -18295.3,E2 -18295.3} C_VEL
LIN {X 0,Y 263.137,Z 902.518,A -85,B 0,C 180,E1 -18298.735,E2 -18298.735} C_VEL
